REGION Network 6: Set SafetyGate Lock
   // 安全门锁定
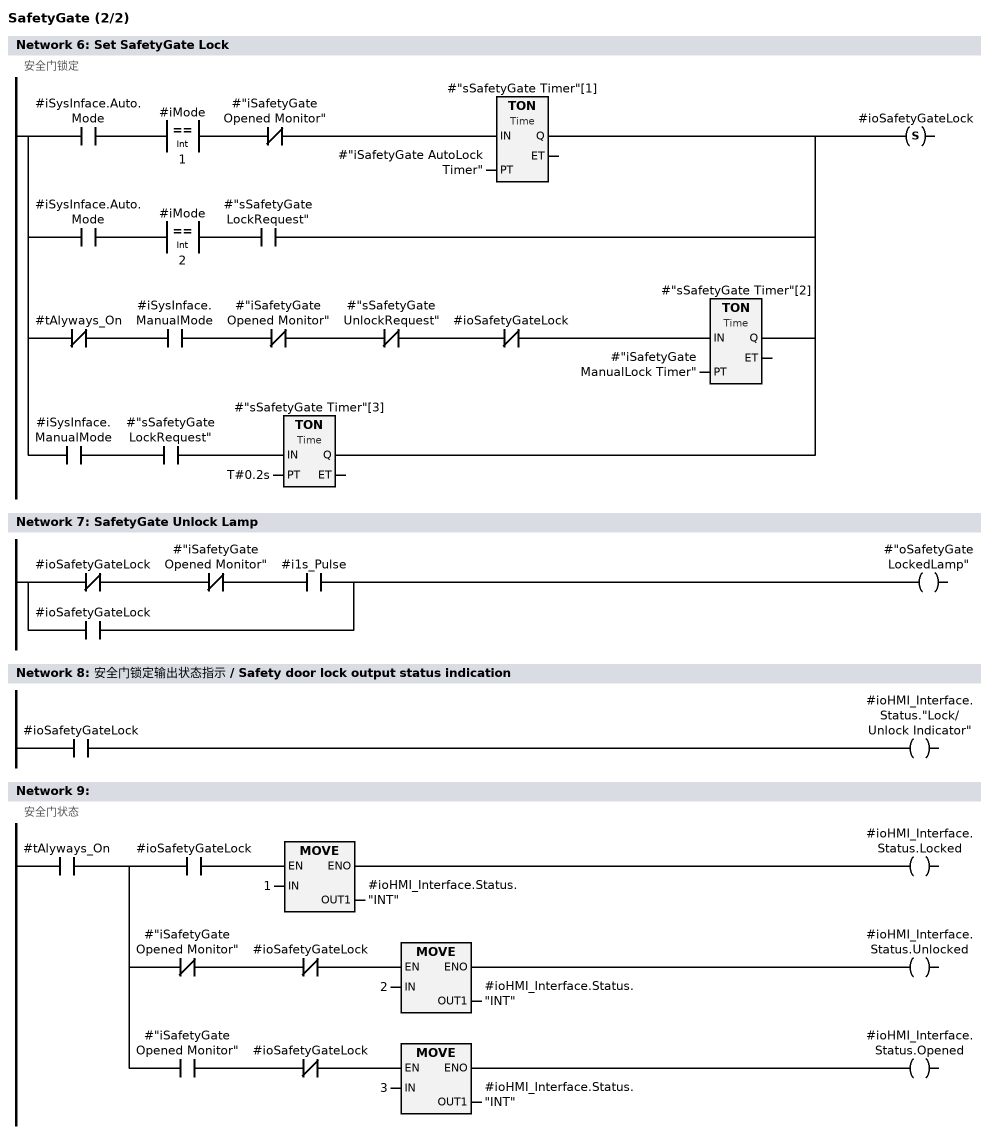
   RUNG wire#powerrail
      Contact( #iSysInface.Auto.Mode )
      { S7_Templates := "SrcType := Int" } EQ_Contact(in1 := #iMode, in2 := 1)
      I_Contact( #"iSafetyGate Opened Monitor" )
      { S7_Templates := "time_type := Time" } #"sSafetyGate Timer"[1].TON(pt := #"iSafetyGate AutoLock Timer", et =>)
      wire#w1
      S_Coil( #ioSafetyGateLock )
   END_RUNG
   RUNG wire#powerrail
      Contact( #iSysInface.Auto.Mode )
      { S7_Templates := "SrcType := Int" } EQ_Contact(in1 := #iMode, in2 := 2)
      Contact( #"sSafetyGate LockRequest" )
   END_RUNG wire#w1
   RUNG wire#powerrail
      I_Contact( #tAlyways_On )
      Contact( #iSysInface.ManualMode )
      I_Contact( #"iSafetyGate Opened Monitor" )
      I_Contact( #"sSafetyGate UnlockRequest" )
      I_Contact( #ioSafetyGateLock )
      { S7_Templates := "time_type := Time" } #"sSafetyGate Timer"[2].TON(pt := #"iSafetyGate ManualLock Timer", et =>)
   END_RUNG wire#w1
   RUNG wire#powerrail
      Contact( #iSysInface.ManualMode )
      Contact( #"sSafetyGate LockRequest" )
      { S7_Templates := "time_type := Time" } #"sSafetyGate Timer"[3].TON(pt := T#0.2s, et =>)
   END_RUNG wire#w1
   // the same network as SCL:
   #"sSafetyGate Timer"[1].TON(IN := #iSysInface.Auto.Mode AND (#iMode = 1) AND NOT #"iSafetyGate Opened Monitor",
                           PT := #"iSafetyGate AutoLock Timer");
   #_w1 := #"sSafetyGate Timer"[1].Q;
   #"sSafetyGate Timer"[2].TON(IN := NOT #tAlyways_On AND #iSysInface.ManualMode AND NOT #"iSafetyGate Opened Monitor" AND NOT #"sSafetyGate UnlockRequest" AND NOT #ioSafetyGateLock,
                           PT := #"iSafetyGate ManualLock Timer");
   #_w2 := #"sSafetyGate Timer"[2].Q;
   #"sSafetyGate Timer"[3].TON(IN := #iSysInface.ManualMode AND #"sSafetyGate LockRequest", PT := T#0.2s);
   IF #_w1 OR (#iSysInface.Auto.Mode AND (#iMode = 2) AND #"sSafetyGate LockRequest") OR #_w2 OR #"sSafetyGate Timer"[3].Q THEN
       #ioSafetyGateLock := TRUE;
   END_IF;
END_REGION

REGION Network 7: SafetyGate Unlock Lamp
   RUNG wire#powerrail
      I_Contact( #ioSafetyGateLock )
      I_Contact( #"iSafetyGate Opened Monitor" )
      Contact( #i1s_Pulse )
      wire#w1
      Coil( #"oSafetyGate LockedLamp" )
   END_RUNG
   RUNG wire#powerrail
      Contact( #ioSafetyGateLock )
   END_RUNG wire#w1
   // the same network as SCL:
   #"oSafetyGate LockedLamp" := (NOT #ioSafetyGateLock AND NOT #"iSafetyGate Opened Monitor" AND #i1s_Pulse) OR #ioSafetyGateLock;
END_REGION

REGION Network 8: 安全门锁定输出状态指示 / Safety door lock output status indication
   RUNG wire#powerrail
      Contact( #ioSafetyGateLock )
      Coil( #ioHMI_Interface.Status."Lock/Unlock Indicator" )
   END_RUNG
   // the same network as SCL:
   #ioHMI_Interface.Status."Lock/Unlock Indicator" := #ioSafetyGateLock;
END_REGION

REGION Network 9
   // 安全门状态
   RUNG wire#powerrail
      Contact( #tAlyways_On )
      wire#w1
      Contact( #ioSafetyGateLock )
      Move(in := 1, out1 => #ioHMI_Interface.Status."INT")
      Coil( #ioHMI_Interface.Status.Locked )
   END_RUNG
   RUNG wire#w1
      I_Contact( #"iSafetyGate Opened Monitor" )
      I_Contact( #ioSafetyGateLock )
      Move(in := 2, out1 => #ioHMI_Interface.Status."INT")
      Coil( #ioHMI_Interface.Status.Unlocked )
   END_RUNG
   RUNG wire#w1
      Contact( #"iSafetyGate Opened Monitor" )
      I_Contact( #ioSafetyGateLock )
      Move(in := 3, out1 => #ioHMI_Interface.Status."INT")
      Coil( #ioHMI_Interface.Status.Opened )
   END_RUNG
   // the same network as SCL:
   #_w1 := #tAlyways_On AND #ioSafetyGateLock;
   IF #_w1 THEN #ioHMI_Interface.Status."INT" := 1; END_IF;
   #ioHMI_Interface.Status.Locked := #_w1;
   #_w2 := #tAlyways_On AND NOT #"iSafetyGate Opened Monitor" AND NOT #ioSafetyGateLock;
   IF #_w2 THEN #ioHMI_Interface.Status."INT" := 2; END_IF;
   #ioHMI_Interface.Status.Unlocked := #_w2;
   #_w3 := #tAlyways_On AND #"iSafetyGate Opened Monitor" AND NOT #ioSafetyGateLock;
   IF #_w3 THEN #ioHMI_Interface.Status."INT" := 3; END_IF;
   #ioHMI_Interface.Status.Opened := #_w3;
END_REGION
END_FUNCTION_BLOCK

FUNCTION "ST10_PartData" : Void   // FC1500, SCL
{ S7_Optimized_Access := 'TRUE' }
// stored: SetENOAutomatically false
   VAR_INPUT
      iSysMode : "RCS_SysComInterface_V1";
   END_VAR
   VAR_TEMP
      idex : Int;
   END_VAR
BEGIN
END_FUNCTION

FUNCTION "ST10_Analog" : Void   // FC1080, SCL
{ S7_Optimized_Access := 'TRUE' }
// stored: AutoNumber false, SetENOAutomatically false
   VAR_INPUT
      iSysMode : "RCS_SysComInterface_V1";
   END_VAR
   VAR_TEMP
      idex : Int;
   END_VAR
BEGIN


   REGION 氮气压模拟量
       //定义编号
       #idex := 1;
       //功能块调用

    END_REGION
END_FUNCTION

FUNCTION "CuringOven" : Void   // FC900, LAD
{ S7_Optimized_Access := 'TRUE' }
// stored: AutoNumber false, SetENOAutomatically false
BEGIN

REGION Network 1
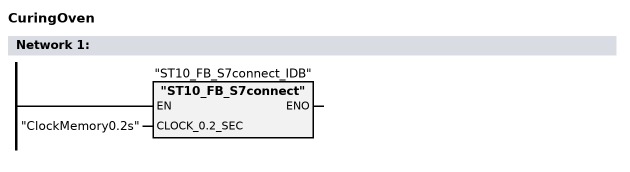
   RUNG wire#powerrail
      "ST10_FB_S7connect_IDB"("CLOCK_0.2_SEC" := "ClockMemory0.2s")
   END_RUNG
   // the same network as SCL:
   "ST10_FB_S7connect_IDB"("CLOCK_0.2_SEC" := "ClockMemory0.2s");   // "ST10_FB_S7connect"
END_REGION
END_FUNCTION

FUNCTION_BLOCK "ST10_FB_S7connect"   // FB900, LAD
{ S7_Optimized_Access := 'TRUE' }
VERSION : 0.1
// stored: AutoNumber false, IsIECCheckEnabled false, IsRetainMemResEnabled false, MemoryReserve 100, SetENOAutomatically false, UDAEnableTagReadback false
   VAR_INPUT
      "CLOCK_0.2_SEC" : Bool;
   END_VAR
   VAR
      Always_On : Bool;
      Status_Get : Array[1..6] of Struct
         NDR : Bool;
         Error : Bool;
         Status : Int;
      END_STRUCT;
      Status_Put : Array[1..6] of Struct
         Done : Bool;
         Error : Bool;
         Status : Int;
      END_STRUCT;
      GET_Instance1 { S7_SetPoint := 'True'} : GET;
      GET_Instance2 { S7_SetPoint := 'True'} : GET;
      PUT_Instance1 { S7_SetPoint := 'True'} : PUT;
      PUT_Instance2 { S7_SetPoint := 'True'} : PUT;
      PLs { S7_SetPoint := 'True'} : Array[1..6] of Bool;
   END_VAR
   VAR DB_SPECIFIC
      TON : Array[1..5] of TON_TIME;
   END_VAR
   VAR
      NextStation_OffLine : Bool;   // S7心跳超时
   END_VAR
BEGIN

REGION Network 1: **************** 和40交互 **************** / **************** ****************
END_REGION

REGION Network 2: PUT
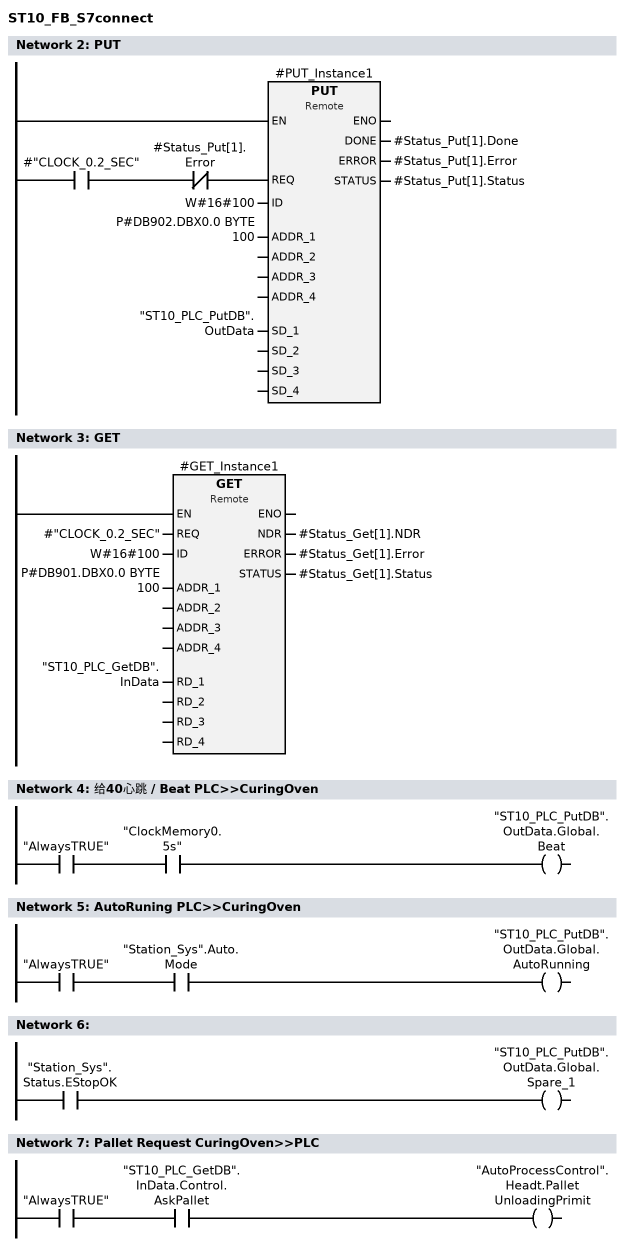
   RUNG wire#powerrail
      { S7_Templates := "[remote_type := Remote, local_type := Variant]" } #PUT_Instance1.PUT(REQ := wire#w1, ID := W#16#100, ADDR_1 := P#DB902.DBX0.0 BYTE 100, ADDR_2 :=, ADDR_3 :=, ADDR_4 :=, SD_1 := "ST10_PLC_PutDB".OutData, SD_2 :=, SD_3 :=, SD_4 :=, DONE => #Status_Put[1].Done, ERROR => #Status_Put[1].Error, STATUS => #Status_Put[1].Status)
   END_RUNG
   RUNG wire#powerrail
      Contact( #"CLOCK_0.2_SEC" )
      I_Contact( #Status_Put[1].Error )
   END_RUNG wire#w1
   // the same network as SCL:
   #PUT_Instance1(REQ := #"CLOCK_0.2_SEC" AND NOT #Status_Put[1].Error,   // PUT
                  ID := W#16#100,
                  ADDR_1 := P#DB902.DBX0.0 BYTE 100,
                  SD_1 := "ST10_PLC_PutDB".OutData,
                  DONE => #Status_Put[1].Done,
                  ERROR => #Status_Put[1].Error,
                  STATUS => #Status_Put[1].Status);
END_REGION

REGION Network 3: GET
   RUNG wire#powerrail
      { S7_Templates := "[remote_type := Remote, local_type := Variant]" } #GET_Instance1.GET(REQ := #"CLOCK_0.2_SEC", ID := W#16#100, ADDR_1 := P#DB901.DBX0.0 BYTE 100, ADDR_2 :=, ADDR_3 :=, ADDR_4 :=, RD_1 := "ST10_PLC_GetDB".InData, RD_2 :=, RD_3 :=, RD_4 :=, NDR => #Status_Get[1].NDR, ERROR => #Status_Get[1].Error, STATUS => #Status_Get[1].Status)
   END_RUNG
   // the same network as SCL:
   #GET_Instance1(REQ := #"CLOCK_0.2_SEC",   // GET
                  ID := W#16#100,
                  ADDR_1 := P#DB901.DBX0.0 BYTE 100,
                  RD_1 := "ST10_PLC_GetDB".InData,
                  NDR => #Status_Get[1].NDR,
                  ERROR => #Status_Get[1].Error,
                  STATUS => #Status_Get[1].Status);
END_REGION

REGION Network 4: 给40心跳 / Beat PLC>>CuringOven
   RUNG wire#powerrail
      Contact( "AlwaysTRUE" )
      Contact( "ClockMemory0.5s" )
      Coil( "ST10_PLC_PutDB".OutData.Global.Beat )
   END_RUNG
   // the same network as SCL:
   "ST10_PLC_PutDB".OutData.Global.Beat := "AlwaysTRUE" AND "ClockMemory0.5s";
END_REGION

REGION Network 5: AutoRuning PLC>>CuringOven
   RUNG wire#powerrail
      Contact( "AlwaysTRUE" )
      Contact( "Station_Sys".Auto.Mode )
      Coil( "ST10_PLC_PutDB".OutData.Global.AutoRunning )
   END_RUNG
   // the same network as SCL:
   "ST10_PLC_PutDB".OutData.Global.AutoRunning := "AlwaysTRUE" AND "Station_Sys".Auto.Mode;
END_REGION

REGION Network 6
   RUNG wire#powerrail
      Contact( "Station_Sys".Status.EStopOK )
      Coil( "ST10_PLC_PutDB".OutData.Global.Spare_1 )
   END_RUNG
   // the same network as SCL:
   "ST10_PLC_PutDB".OutData.Global.Spare_1 := "Station_Sys".Status.EStopOK;
END_REGION

REGION Network 7: Pallet Request CuringOven>>PLC
   RUNG wire#powerrail
      Contact( "AlwaysTRUE" )
      Contact( "ST10_PLC_GetDB".InData.Control.AskPallet )
      Coil( "AutoProcessControl".Headt.PalletUnloadingPrimit )
   END_RUNG
   // the same network as SCL:
   "AutoProcessControl".Headt.PalletUnloadingPrimit := "AlwaysTRUE" AND "ST10_PLC_GetDB".InData.Control.AskPallet;
END_REGION
END_FUNCTION_BLOCK

FUNCTION "IV3" : Void   // FC2100, LAD
{ S7_Optimized_Access := 'TRUE' }
VERSION : 0.1
// stored: AutoNumber false, IsIECCheckEnabled false, SetENOAutomatically false, UDAEnableTagReadback false
BEGIN

REGION Network 1: IV3
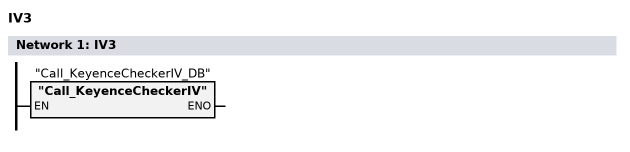
   RUNG wire#powerrail
      "Call_KeyenceCheckerIV_DB"()
   END_RUNG
   // the same network as SCL:
   "Call_KeyenceCheckerIV_DB"();   // "Call_KeyenceCheckerIV"
END_REGION
END_FUNCTION

FUNCTION_BLOCK "Call_KeyenceCheckerIV"   // FB2100, SCL
{ S7_Optimized_Access := 'TRUE' }
// stored: AutoNumber false, MemoryReserve 100, SetENOAutomatically false
   VAR
      InsKeyenceCheckerIV3810A1 : "FB_KeyenceCheckerIV3";   // 声明相机功能块的实例
      InsKeyenceCheckerIV3811A1 : "FB_KeyenceCheckerIV3";   // 声明相机功能块的实例
      nIndex { S7_SetPoint := 'True'} : Int;
   END_VAR
BEGIN

   //810A1
   REGION KeyenceCheckerIV3() 

       REGION HardwareConfigGuidance()
           // 组态说明/Hardware config Guidance
           // 输入/Input
           // Command Status Bits_1
           // Device Result Bits_1
           // Device Status Words_1
           // Device Statistics_1
           // Position Adjust Result_1
           // Tool Result_1
           // Tool Result_2
           // 输出/Output
           // Command Control_1
       END_REGION

       REGION DeviceControl()
           //************************************************************************************************ 
           //设备控制/Device control 
           //************************************************************************************************ 
           //Set device number
           #nIndex := 1;//(For example Constant:ST01_CHECKER_FUNCTION)

           REGION WorkflowControl()
               //************************************************************************************************ 
               //流程控制/Workflow control
               //************************************************************************************************ 
               //---set program number
               //   "DB_KeyenceCheckerIV2".aDev[#nIndex].Out.CommandControl.nProgramNo
               //---set command mode and wait for mode to "MODE_CHECKER_IDLE"
               //   "DB_KeyenceCheckerIV2".aDev[#nIndex].Common.nMode
           END_REGION

           REGION GeneralControl()
               //************************************************************************************************ 
               //常规控制/General control 
               //************************************************************************************************ 
               //Set common parameter
               "DB_KeyenceCheckerIV3".aDev[#nIndex].Common.bScreenActive := "Station_Sys".Manual.Mode;
               "DB_KeyenceCheckerIV3".aDev[#nIndex].Common.bReset := "Station_Sys".Cmd.Reset;
               "DB_KeyenceCheckerIV3".aDev[#nIndex].Common.tMaxProcessTime := t#30s;
           END_REGION

           REGION ParameterConfig()
               //************************************************************************************************ 
               //参数配置/Parameter config 
               //************************************************************************************************ 
           END_REGION

           REGION ModeControl()
               //************************************************************************************************ 
               //设备启动停止/Device mode control
               //************************************************************************************************ 
               // IF NOT "Station_Sys".Status.Run THEN
               //     "DB_KeyenceCheckerIV3".aDev[#nIndex].Common.nMode := 0;
               // END_IF;

               IF "Station_Sys".Manual.Mode THEN
                   "DB_KeyenceCheckerIV3".aDev[#nIndex].Common.nModeSwitch := "MS_MANUAL";
               ELSIF "Station_Sys".Auto.Mode THEN
                   "DB_KeyenceCheckerIV3".aDev[#nIndex].Common.nModeSwitch:=  "MS_Auto";
               ELSE
                   "DB_KeyenceCheckerIV3".aDev[#nIndex].Common.nModeSwitch := "MS_EMPTY";
               END_IF;
               END_REGION

           REGION ConditionControl()
               //************************************************************************************************ 
               //使能控制/Condition control
               //************************************************************************************************ 
               //according to detail information in different use to fill in start condition
               "DB_KeyenceCheckerIV3".aDev[#nIndex].Common.bEnable := "Station_Sys".Status.Run;
           END_REGION

       END_REGION

       REGION HardwareInput()
           //************************************************************************************************ 
           //硬件输入/Hardware input 
           //************************************************************************************************ 
       END_REGION

       REGION CallFunctionBlock()
           //************************************************************************************************
           //功能块调用/Call function block
           //************************************************************************************************
           //according to hardware configuration to type in hardware address

           #InsKeyenceCheckerIV3810A1(#nIndex);


       END_REGION

       REGION HardwareOutput()
           //************************************************************************************************ 
           //硬件输出/Hardware output 
           //************************************************************************************************ 
       END_REGION

   END_REGION


   //811A1
   REGION KeyenceCheckerIV3() 

       REGION HardwareConfigGuidance()
           // 组态说明/Hardware config Guidance
           // 输入/Input
           // Command Status Bits_1
           // Device Result Bits_1
           // Device Status Words_1
           // Device Statistics_1
           // Position Adjust Result_1
           // Tool Result_1
           // Tool Result_2
           // 输出/Output
           // Command Control_1
       END_REGION

       REGION DeviceControl()
           //************************************************************************************************ 
           //设备控制/Device control 
           //************************************************************************************************ 
           //Set device number
           #nIndex := 2;//(For example Constant:ST01_CHECKER_FUNCTION)

           REGION WorkflowControl()
               //************************************************************************************************ 
               //流程控制/Workflow control
               //************************************************************************************************ 
               //---set program number
               //   "DB_KeyenceCheckerIV2".aDev[#nIndex].Out.CommandControl.nProgramNo
               //---set command mode and wait for mode to "MODE_CHECKER_IDLE"
               //   "DB_KeyenceCheckerIV2".aDev[#nIndex].Common.nMode
           END_REGION

           REGION GeneralControl()
               //************************************************************************************************ 
               //常规控制/General control 
               //************************************************************************************************ 
               //Set common parameter
               "DB_KeyenceCheckerIV3".aDev[#nIndex].Common.bScreenActive := "Station_Sys".Manual.Mode;
               "DB_KeyenceCheckerIV3".aDev[#nIndex].Common.bReset := "Station_Sys".Cmd.Reset;
               "DB_KeyenceCheckerIV3".aDev[#nIndex].Common.tMaxProcessTime := t#30s;
           END_REGION

           REGION ParameterConfig()
               //************************************************************************************************ 
               //参数配置/Parameter config 
               //************************************************************************************************ 
           END_REGION

           REGION ModeControl()
               //************************************************************************************************ 
               //设备启动停止/Device mode control
               //************************************************************************************************ 
               // IF NOT "Station_Sys".Status.Run THEN
               //     "DB_KeyenceCheckerIV3".aDev[#nIndex].Common.nMode := 0;
               // END_IF;

               IF "Station_Sys".Manual.Mode THEN
                   "DB_KeyenceCheckerIV3".aDev[#nIndex].Common.nModeSwitch := "MS_MANUAL";
               ELSIF "Station_Sys".Auto.Mode THEN
                   "DB_KeyenceCheckerIV3".aDev[#nIndex].Common.nModeSwitch := "MS_Auto";
               ELSE
                   "DB_KeyenceCheckerIV3".aDev[#nIndex].Common.nModeSwitch := "MS_EMPTY";
               END_IF;
           END_REGION

           REGION ConditionControl()
               //************************************************************************************************ 
               //使能控制/Condition control
               //************************************************************************************************ 
               //according to detail information in different use to fill in start condition
               "DB_KeyenceCheckerIV3".aDev[#nIndex].Common.bEnable := "Station_Sys".Status.Run;
           END_REGION

       END_REGION

       REGION HardwareInput()
           //************************************************************************************************ 
           //硬件输入/Hardware input 
           //************************************************************************************************ 
       END_REGION

       REGION CallFunctionBlock()
           //************************************************************************************************
           //功能块调用/Call function block
           //************************************************************************************************
           //according to hardware configuration to type in hardware address

           #InsKeyenceCheckerIV3811A1(#nIndex);


       END_REGION

       REGION HardwareOutput()
           //************************************************************************************************ 
           //硬件输出/Hardware output 
           //************************************************************************************************ 
       END_REGION

   END_REGION
END_FUNCTION_BLOCK

FUNCTION "IAI" : Void   // FC2200, LAD
{ S7_Optimized_Access := 'TRUE' }
// stored: AutoNumber false, SetENOAutomatically false
BEGIN

REGION Network 1 (SCL): 模式 / Mode
   "ModeDB".Gen.Out.Estop := "Station_Sys".Status.EStopOK;
   "ModeDB".Gen.Out.Reset := "Station_Sys".Cmd.Reset;
   "ModeDB".Gen.Out.Manual := "Station_Sys".Manual.Mode;
   "ModeDB".Gen.Out.Auto := "Station_Sys".Auto.Mode;
   "ModeDB".Gen.Out.Home := "Station_Sys".Initial.Running;
   "ModeDB".Gen.Out.Running := "Station_Sys".Auto.Mode;//"Station_Sys".Auto.Running OR "ST10_PM".Num[7].InitialRun;
   //"ModeDB".Gen.Out.Change:=
END_REGION

REGION Network 2
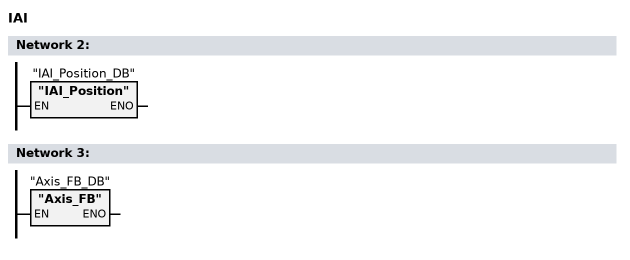
   RUNG wire#powerrail
      "IAI_Position_DB"()
   END_RUNG
   // the same network as SCL:
   "IAI_Position_DB"();   // "IAI_Position"
END_REGION

REGION Network 3
   RUNG wire#powerrail
      "Axis_FB_DB"()
   END_RUNG
   // the same network as SCL:
   "Axis_FB_DB"();   // "Axis_FB"
END_REGION
END_FUNCTION

FUNCTION_BLOCK "IAI_Position"   // FB2210, LAD
{ S7_Optimized_Access := 'TRUE' }
// stored: AutoNumber false, MemoryReserve 100, SetENOAutomatically false
   VAR
      Servo5 { S7_SetPoint := 'True'} : "SevroStart&PosCheck_IAI";
      Servo6 { S7_SetPoint := 'True'} : "SevroStart&PosCheck_IAI";
      Servo7 { S7_SetPoint := 'True'} : "SevroStart&PosCheck_IAI";
   END_VAR
   VAR_TEMP
      Sevro5ActPos : Real;
      Sevro5StartList : Bool;
      Sevro6ActPos : Real;
      Sevro6StartList : Bool;
      Sevro7ActPos : Real;
      Sevro7StartList : Bool;
   END_VAR
BEGIN

REGION Network 2 (SCL)
   REGION Servo position judgment
       FOR "IAI_DeviceCtl".IAIServo[1].i := 1 TO 12 BY 1 DO
           "IAI_DeviceCtl".IAIServo[1].Pos.List["IAI_DeviceCtl".IAIServo[1].i].Pos := "IAI_A1".Auto.Pos["IAI_DeviceCtl".IAIServo[1].i].Pos;
           "IAI_DeviceCtl".IAIServo[1].Pos.List["IAI_DeviceCtl".IAIServo[1].i].Vel := "IAI_A1".Auto.Pos["IAI_DeviceCtl".IAIServo[1].i].Vel;

           "IAI_DeviceCtl".IAIServo[2].Pos.List["IAI_DeviceCtl".IAIServo[1].i].Pos := "IAI_A2".Auto.Pos["IAI_DeviceCtl".IAIServo[1].i].Pos;
           "IAI_DeviceCtl".IAIServo[2].Pos.List["IAI_DeviceCtl".IAIServo[1].i].Vel := "IAI_A2".Auto.Pos["IAI_DeviceCtl".IAIServo[1].i].Vel;

           "IAI_DeviceCtl".IAIServo[3].Pos.List["IAI_DeviceCtl".IAIServo[1].i].Pos := "IAI_A3".Auto.Pos["IAI_DeviceCtl".IAIServo[1].i].Pos;
           "IAI_DeviceCtl".IAIServo[3].Pos.List["IAI_DeviceCtl".IAIServo[1].i].Vel := "IAI_A3".Auto.Pos["IAI_DeviceCtl".IAIServo[1].i].Vel;


       END_FOR;

       (******************************************************* SV1 Z轴 ********************************************************************)
       //伺服位置判断
       #"Servo5"(iRef_Homed := 1,
                 iStandstill := FALSE,
                 iReset := "Station_Sys".Cmd.Reset,
                 interlcok := 1,
                 "iActual Posi" := "Axis_FB_DB".IAI_Axis[1].CurrentPosition,
                 "iTol+" := 0.5,
                 "iTol-" := 0.5,
                 iStartTon := T#100mS,
                 ioPoint := "IAI_DeviceCtl".IAIServo[1].Point,
                 oStartPos => #Sevro5StartList,
                 ioList := "IAI_DeviceCtl".IAIServo[1].Pos,
                 ioPosNumberSelect := "IAI_DeviceCtl".IAIServo[1].nPositionListNo);

       IF "IAI_DeviceCtl".IAIServo[1].nPositionListNo = 0 THEN
           "IAI_DeviceCtl".IAIServo[1].nPositionListNo := 1;
       END_IF;

       "Axis_FB_DB".IAI_Axis[1].Par.PosCode:="IAI_A1".Auto.Index := "IAI_DeviceCtl".IAIServo[1].nPositionListNo;

       //伺服启动
       "IAI_A1".In.iAutoStart := #Sevro5StartList AND "Station_Sys".Auto.Mode;

       (******************************************************* SV2 X轴********************************************************************)
       //伺服位置判断
       #"Servo6"(iRef_Homed := 1,
                 iStandstill := FALSE,
                 iReset := "Station_Sys".Cmd.Reset,
                 interlcok := 1,
                 "iActual Posi" := "Axis_FB_DB".IAI_Axis[2].CurrentPosition,
                 "iTol+" := 0.5,
                 "iTol-" := 0.5,
                 iStartTon := T#100mS,
                 ioPoint := "IAI_DeviceCtl".IAIServo[2].Point,
                 oStartPos => #Sevro6StartList,
                 ioList := "IAI_DeviceCtl".IAIServo[2].Pos,
                 ioPosNumberSelect := "IAI_DeviceCtl".IAIServo[2].nPositionListNo);

       IF "IAI_DeviceCtl".IAIServo[2].nPositionListNo = 0 THEN
           "IAI_DeviceCtl".IAIServo[2].nPositionListNo := 1;
       END_IF;

       "Axis_FB_DB".IAI_Axis[2].Par.PosCode:="IAI_A2".Auto.Index := "IAI_DeviceCtl".IAIServo[2].nPositionListNo;

       //伺服启动
       "IAI_A2".In.iAutoStart := #Sevro6StartList AND "Station_Sys".Auto.Mode;

       (******************************************************* SV3 Y轴********************************************************************)
       //伺服位置判断
       #"Servo7"(iRef_Homed := 1,
                 iStandstill := FALSE,
                 iReset := "Station_Sys".Cmd.Reset,
                 interlcok := 1,
                 "iActual Posi" := "Axis_FB_DB".IAI_Axis[3].CurrentPosition,
                 "iTol+" := 0.5,
                 "iTol-" := 0.5,
                 iStartTon := T#100mS,
                 ioPoint := "IAI_DeviceCtl".IAIServo[3].Point,
                 oStartPos => #Sevro7StartList,
                 ioList := "IAI_DeviceCtl".IAIServo[3].Pos,
                 ioPosNumberSelect := "IAI_DeviceCtl".IAIServo[3].nPositionListNo);

       IF "IAI_DeviceCtl".IAIServo[3].nPositionListNo = 0 THEN
           "IAI_DeviceCtl".IAIServo[3].nPositionListNo := 1;
       END_IF;

       "Axis_FB_DB".IAI_Axis[3].Par.PosCode:="IAI_A3".Auto.Index := "IAI_DeviceCtl".IAIServo[3].nPositionListNo;

       //伺服启动
       "IAI_A3".In.iAutoStart := #Sevro7StartList AND "Station_Sys".Auto.Mode;
   END_REGION
END_REGION
END_FUNCTION_BLOCK

FUNCTION_BLOCK "SevroStart&PosCheck_IAI"   // FB2209, LAD
{ S7_Optimized_Access := 'TRUE' }
// stored: AutoNumber false, MemoryReserve 100, SetENOAutomatically false
   VAR_INPUT
      iRef_Homed { ExternalAccessible := 'False'; ExternalVisible := 'False'; ExternalWritable := 'False'} : Bool;
      iStandstill { ExternalAccessible := 'False'; ExternalVisible := 'False'; ExternalWritable := 'False'} : Bool;
      iReset : Bool;
      interlcok : Bool;   // 启动互锁
      "iActual Posi" { ExternalAccessible := 'False'; ExternalVisible := 'False'; ExternalWritable := 'False'} : Real;
      "iTol+" { ExternalAccessible := 'False'; ExternalVisible := 'False'; ExternalWritable := 'False'} : Real;
      "iTol-" { ExternalAccessible := 'False'; ExternalVisible := 'False'; ExternalWritable := 'False'} : Real;
      iStartTon : Time := T#200ms;   // 启动延迟
   END_VAR
   VAR_OUTPUT
      oStartPos : Bool;   // 启动
      DoublePosError : Bool;   // 多位置触发
   END_VAR
   VAR_IN_OUT
      ioPoint : Array[0..39] of Struct
         Start : Bool;
         Achieve : Bool;
      END_STRUCT;
      ioList : "PosList_IAI";
      ioPosNumberSelect : Int;   // 位置启动
   END_VAR
   VAR
      TON : Array[0..1] of TON_TIME;
      StartCount { S7_SetPoint := 'True'} : Int;   // 启动计数
   END_VAR
   VAR_TEMP
      "Actual Posi+Tol" : Real;
      "Actual Posi-Tol" : Real;
      Index : Array[0..7] of Int;   // 位置启动
      PosStart : Bool;
   END_VAR
   VAR_TEMP   // added for the SCL form of the ladder/FBD networks
      _w1 : Bool;
   END_VAR
BEGIN

REGION Network 1 (SCL): 检查当前启动位置号
   #Index[1] := 0;
   #PosStart := false;
   FOR #Index[1] := 0 TO 39 DO
       IF #ioPoint[#Index[1]].Start THEN

           #ioPosNumberSelect := #Index[1];//当前启动位置号
           #PosStart := TRUE;
           EXIT;
       END_IF;
   END_FOR;
   #Index[2] := 0;
   #StartCount := 0;
   FOR #Index[2] := 0 TO 39 DO
       IF #ioPoint[#Index[2]].Start THEN

           #StartCount := #StartCount+1;//当前启动位置号


       END_IF;
       IF #Index[2] = 39 THEN

           EXIT;
       END_IF;

   END_FOR;
END_REGION

REGION Network 2: 位置给定
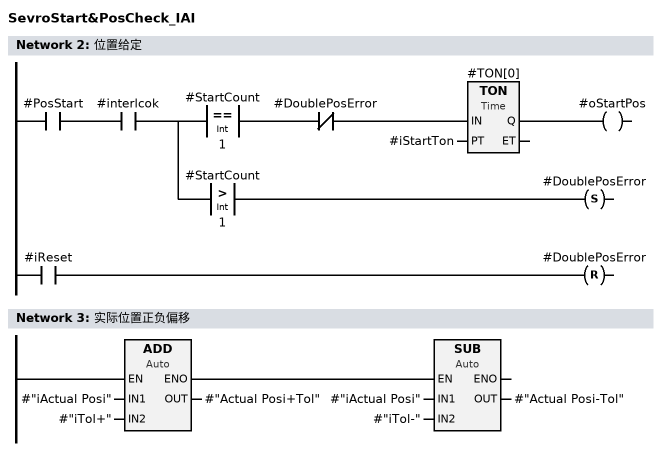
   RUNG wire#powerrail
      Contact( #PosStart )
      Contact( #interlcok )
      wire#w1
      { S7_Templates := "SrcType := Int" } EQ_Contact(in1 := #StartCount, in2 := 1)
      I_Contact( #DoublePosError )
      { S7_Templates := "time_type := Time" } #TON[0].TON(pt := #iStartTon, et =>)
      Coil( #oStartPos )
   END_RUNG
   RUNG wire#w1
      { S7_Templates := "SrcType := Int" } GT_Contact(in1 := #StartCount, in2 := 1)
      S_Coil( #DoublePosError )
   END_RUNG
   RUNG wire#powerrail
      Contact( #iReset )
      R_Coil( #DoublePosError )
   END_RUNG
   // the same network as SCL:
   #_w1 := #PosStart AND #interlcok;
   #TON[0].TON(IN := #_w1 AND (#StartCount = 1) AND NOT #DoublePosError, PT := #iStartTon);
   #oStartPos := #TON[0].Q;
   IF #_w1 AND (#StartCount > 1) THEN #DoublePosError := TRUE; END_IF;
   IF #iReset THEN #DoublePosError := FALSE; END_IF;
END_REGION

REGION Network 3: 实际位置正负偏移
   RUNG wire#powerrail
      Add(in1 := #"iActual Posi", in2 := #"iTol+", out => #"Actual Posi+Tol")
      Sub(in1 := #"iActual Posi", in2 := #"iTol-", out => #"Actual Posi-Tol")
   END_RUNG
   // the same network as SCL:
   #"Actual Posi+Tol" := #"iActual Posi" + #"iTol+";
   #"Actual Posi-Tol" := #"iActual Posi" - #"iTol-";
END_REGION

REGION Network 4 (SCL): 位置检查


   #Index[3] := 0;
   FOR #Index[3] := 0 TO 39 DO
       IF #ioList.List[ #Index[3]].Pos>= #"Actual Posi-Tol"
           AND #ioList.List[ #Index[3]].Pos<= #"Actual Posi+Tol"
       THEN
         #ioPoint[#Index[3]].Achieve := TRUE;
       ELSE
           #ioPoint[#Index[3]].Achieve := FALSE;
       END_IF;
   END_FOR;
END_REGION
END_FUNCTION_BLOCK

FUNCTION_BLOCK "Axis_FB"   // FB2200, SCL
{ S7_Optimized_Access := 'FALSE' }
// stored: AutoNumber false, SetENOAutomatically false
   VAR
      IAI_Axis { S7_SetPoint := 'True'} : Array[1..3] of "IAI_BASE_FB";
   END_VAR
   VAR CONSTANT
      Z_Axis : Int := 1;
      Y_axis : Int := 3;
      X_Axis : Int := 2;
   END_VAR
BEGIN
   ///Z轴

   #IAI_Axis[X_Axis].Enable := #IAI_Axis[Y_axis].Enable := #IAI_Axis[Z_Axis].Enable := "ST10_SystemModeFB_iDB".iEstopAllOK AND "ST10_SystemModeFB_iDB".iSafetyDoor;

   #IAI_Axis[Z_Axis]();

   #IAI_Axis[Z_Axis].Axis_ID := 1;
   #IAI_Axis[Z_Axis]."Input 4 word_Man1" := "OP10_384A1~Input_4_word_7";
   #IAI_Axis[Z_Axis]."Input 4 word_Man2" := "OP10_384A1~Input_4_word_8";
   #IAI_Axis[Z_Axis]."Input 4 word_1" := "OP10_384A1~Input_4_word_3";
   #IAI_Axis[Z_Axis]."Input 4 word_2" := "OP10_384A1~Input_4_word_4";
   #IAI_Axis[Z_Axis]."Output 4 word_Man1" := "OP10_384A1~Output_4_word_1";
   #IAI_Axis[Z_Axis]."Output 4 word_Man2" := "OP10_384A1~Output_4_word_2";
   #IAI_Axis[Z_Axis]."Output 4 word_1" := "OP10_384A1~Output_4_word_5";
   #IAI_Axis[Z_Axis]."Output 4 word_2" := "OP10_384A1~Output_4_word_6";

   #IAI_Axis[Z_Axis].Mode:= "ModeDB".Gen;
   #IAI_Axis[Z_Axis].Par.PositionWidth := 0.05;
   #IAI_Axis[Z_Axis].Par.AccSpeed := 10;
   #IAI_Axis[Z_Axis].Par.DecSpeed := 10;
   #IAI_Axis[Z_Axis].Par."Limt+Pos" := 362000.0;
   #IAI_Axis[Z_Axis].Par."Limt-Pos" := -30000.0;
   #IAI_Axis[Z_Axis].Par.Speed:= 10;

   #IAI_Axis[Z_Axis].Interfere := TRUE;
   #IAI_Axis[Z_Axis].RunSetTime := T#20S;
   #IAI_Axis[Z_Axis].Par.GoPosInterfere[0] := TRUE;
   #IAI_Axis[Z_Axis].Par.GoPosInterfere[1] := TRUE;
   #IAI_Axis[Z_Axis].Par.GoPosInterfere[2] := TRUE;
   #IAI_Axis[Z_Axis].Par.GoPosInterfere[3] := TRUE;
   #IAI_Axis[Z_Axis].Par.GoPosInterfere[4] := TRUE;
   #IAI_Axis[Z_Axis].Par.GoPosInterfere[5] := TRUE;
   #IAI_Axis[Z_Axis].AutoPointStart := "IAI_A1".In.iAutoStart;

   "IAI_A1".Auto.Pos[1].Pos:=#IAI_Axis[Z_Axis].Par.TargetPosition[1] := "Parameter".AxisRun.Axis[5].Pos1.Position;
   "IAI_A1".Auto.Pos[1].Vel :=#IAI_Axis[Z_Axis].Par.TargetSpeed[1] := "Parameter".AxisRun.Axis[5].Pos1.Speed;

   "IAI_A1".Auto.Pos[2].Pos:=#IAI_Axis[Z_Axis].Par.TargetPosition[2] := "Parameter".AxisRun.Axis[5].Pos2.Position;
   "IAI_A1".Auto.Pos[2].Vel :=#IAI_Axis[Z_Axis].Par.TargetSpeed[2] := "Parameter".AxisRun.Axis[5].Pos2.Speed;

   "IAI_A1".Auto.Pos[3].Pos:=#IAI_Axis[Z_Axis].Par.TargetPosition[3] := "Parameter".AxisRun.Axis[5].Pos3.Position;
   "IAI_A1".Auto.Pos[3].Vel :=#IAI_Axis[Z_Axis].Par.TargetSpeed[3] := "Parameter".AxisRun.Axis[5].Pos3.Speed;

   "IAI_A1".Auto.Pos[4].Pos:=#IAI_Axis[Z_Axis].Par.TargetPosition[4] := "Parameter".AxisRun.Axis[5].Pos4.Position;
   "IAI_A1".Auto.Pos[4].Vel :=#IAI_Axis[Z_Axis].Par.TargetSpeed[4] := "Parameter".AxisRun.Axis[5].Pos4.Speed;

   "IAI_A1".Auto.Pos[5].Pos:=#IAI_Axis[Z_Axis].Par.TargetPosition[5] := "Parameter".AxisRun.Axis[5].Pos5.Position;
   "IAI_A1".Auto.Pos[5].Vel :=#IAI_Axis[Z_Axis].Par.TargetSpeed[5] := "Parameter".AxisRun.Axis[5].Pos5.Speed;

   "IAI_A1".Auto.Pos[6].Pos := #IAI_Axis[Z_Axis].Par.TargetPosition[6] := "Parameter".AxisRun.Axis[5].Pos6.Position;
   "IAI_A1".Auto.Pos[6].Vel := #IAI_Axis[Z_Axis].Par.TargetSpeed[6] := "Parameter".AxisRun.Axis[5].Pos6.Speed;

   "IAI_A1".Auto.Pos[7].Pos := #IAI_Axis[Z_Axis].Par.TargetPosition[7] := "Parameter".AxisRun.Axis[5].Pos7.Position;
   "IAI_A1".Auto.Pos[7].Vel := #IAI_Axis[Z_Axis].Par.TargetSpeed[7] := "Parameter".AxisRun.Axis[5].Pos7.Speed;

   "IAI_A1".Auto.Pos[8].Pos := #IAI_Axis[Z_Axis].Par.TargetPosition[8] := "Parameter".AxisRun.Axis[5].Pos8.Position;
   "IAI_A1".Auto.Pos[8].Vel := #IAI_Axis[Z_Axis].Par.TargetSpeed[8] := "Parameter".AxisRun.Axis[5].Pos8.Speed;

   "IAI_A1".Auto.Pos[9].Pos := #IAI_Axis[Z_Axis].Par.TargetPosition[9] := "Parameter".AxisRun.Axis[5].Pos6.Position-4.0;
   "IAI_A1".Auto.Pos[9].Vel := #IAI_Axis[Z_Axis].Par.TargetSpeed[9] := "Parameter".AxisRun.Axis[5].Pos6.Speed;

   "IAI_A1".Auto.Pos[10].Pos := #IAI_Axis[Z_Axis].Par.TargetPosition[10] := "Parameter".AxisRun.Axis[5].Pos10.Position;
   "IAI_A1".Auto.Pos[10].Vel := #IAI_Axis[Z_Axis].Par.TargetSpeed[10] := "Parameter".AxisRun.Axis[5].Pos10.Speed;

   //X轴
   #IAI_Axis[X_Axis]();

   #IAI_Axis[X_Axis].Axis_ID := 2;
   #IAI_Axis[X_Axis]."Input 4 word_Man1" := "OP10_384A1~Input_4_word_7";
   #IAI_Axis[X_Axis]."Input 4 word_Man2" := "OP10_384A1~Input_4_word_8";
   #IAI_Axis[X_Axis]."Input 4 word_1" := "OP10_384A1~Input_4_word_5";
   #IAI_Axis[X_Axis]."Input 4 word_2" := "OP10_384A1~Input_4_word_6";
   #IAI_Axis[X_Axis]."Output 4 word_Man1" := "OP10_384A1~Output_4_word_1";
   #IAI_Axis[X_Axis]."Output 4 word_Man2" := "OP10_384A1~Output_4_word_2";
   #IAI_Axis[X_Axis]."Output 4 word_1" := "OP10_384A1~Output_4_word_7";
   #IAI_Axis[X_Axis]."Output 4 word_2" := "OP10_384A1~Output_4_word_8";

   #IAI_Axis[X_Axis].Mode := "ModeDB".Gen;
   #IAI_Axis[X_Axis].Par.PositionWidth := 0.05;
   #IAI_Axis[X_Axis].Par.AccSpeed := 10;
   #IAI_Axis[X_Axis].Par.DecSpeed := 10;

   #IAI_Axis[X_Axis].Par."Limt+Pos" := 362000.0;
   #IAI_Axis[X_Axis].Par."Limt-Pos" := -30000.0;
   #IAI_Axis[X_Axis].Interfere := TRUE;
   #IAI_Axis[X_Axis].RunSetTime := T#20S;
   #IAI_Axis[X_Axis].Par.GoPosInterfere[0] := TRUE;
   #IAI_Axis[X_Axis].Par.GoPosInterfere[1] := TRUE;
   #IAI_Axis[X_Axis].Par.GoPosInterfere[2] := TRUE;
   #IAI_Axis[X_Axis].Par.GoPosInterfere[3] := TRUE;
   #IAI_Axis[X_Axis].Par.GoPosInterfere[4] := TRUE;
   #IAI_Axis[X_Axis].Par.GoPosInterfere[5] := TRUE;
   #IAI_Axis[X_Axis].AutoPointStart := "IAI_A2".In.iAutoStart;

   "IAI_A2".Auto.Pos[1].Pos:=#IAI_Axis[X_Axis].Par.TargetPosition[1] := "Parameter".AxisRun.Axis[6].Pos1.Position;
   "IAI_A2".Auto.Pos[1].Vel := #IAI_Axis[X_Axis].Par.TargetSpeed[1] := "Parameter".AxisRun.Axis[6].Pos1.Speed;

   "IAI_A2".Auto.Pos[2].Pos:=#IAI_Axis[X_Axis].Par.TargetPosition[2] := "Parameter".AxisRun.Axis[6].Pos2.Position;
   "IAI_A2".Auto.Pos[2].Vel :=#IAI_Axis[X_Axis].Par.TargetSpeed[2] := "Parameter".AxisRun.Axis[6].Pos2.Speed;

   "IAI_A2".Auto.Pos[3].Pos:=#IAI_Axis[X_Axis].Par.TargetPosition[3] := "Parameter".AxisRun.Axis[6].Pos3.Position;
   "IAI_A2".Auto.Pos[3].Vel :=#IAI_Axis[X_Axis].Par.TargetSpeed[3] := "Parameter".AxisRun.Axis[6].Pos3.Speed;

   "IAI_A2".Auto.Pos[4].Pos:=#IAI_Axis[X_Axis].Par.TargetPosition[4] := "Parameter".AxisRun.Axis[6].Pos4.Position;
   "IAI_A2".Auto.Pos[4].Vel :=#IAI_Axis[X_Axis].Par.TargetSpeed[4] := "Parameter".AxisRun.Axis[6].Pos4.Speed;

   "IAI_A2".Auto.Pos[5].Pos:=#IAI_Axis[X_Axis].Par.TargetPosition[5] := "Parameter".AxisRun.Axis[6].Pos5.Position;
   "IAI_A2".Auto.Pos[5].Vel :=#IAI_Axis[X_Axis].Par.TargetSpeed[5] := "Parameter".AxisRun.Axis[6].Pos5.Speed;

   "IAI_A2".Auto.Pos[6].Pos := #IAI_Axis[X_Axis].Par.TargetPosition[6] := "Parameter".AxisRun.Axis[6].Pos6.Position;
   "IAI_A2".Auto.Pos[6].Vel := #IAI_Axis[X_Axis].Par.TargetSpeed[6] := "Parameter".AxisRun.Axis[6].Pos6.Speed;

   "IAI_A2".Auto.Pos[7].Pos := #IAI_Axis[X_Axis].Par.TargetPosition[7] := "Parameter".AxisRun.Axis[6].Pos7.Position;
   "IAI_A2".Auto.Pos[7].Vel := #IAI_Axis[X_Axis].Par.TargetSpeed[7] := "Parameter".AxisRun.Axis[6].Pos7.Speed;

   "IAI_A2".Auto.Pos[8].Pos := #IAI_Axis[X_Axis].Par.TargetPosition[8] := "Parameter".AxisRun.Axis[6].Pos8.Position;
   "IAI_A2".Auto.Pos[8].Vel := #IAI_Axis[X_Axis].Par.TargetSpeed[8] := "Parameter".AxisRun.Axis[6].Pos8.Speed;

   "IAI_A2".Auto.Pos[9].Pos := #IAI_Axis[X_Axis].Par.TargetPosition[9] := "Parameter".AxisRun.Axis[6].Pos9.Position;
   "IAI_A2".Auto.Pos[9].Vel := #IAI_Axis[X_Axis].Par.TargetSpeed[9] := "Parameter".AxisRun.Axis[6].Pos9.Speed;

   "IAI_A2".Auto.Pos[10].Pos := #IAI_Axis[X_Axis].Par.TargetPosition[10] := "Parameter".AxisRun.Axis[6].Pos10.Position;
   "IAI_A2".Auto.Pos[10].Vel := #IAI_Axis[X_Axis].Par.TargetSpeed[10] := "Parameter".AxisRun.Axis[6].Pos10.Speed;

   ///Y轴
   #IAI_Axis[Y_axis]();

   #IAI_Axis[Y_axis].Axis_ID := 3;
   #IAI_Axis[Y_axis]."Input 4 word_Man1" := "OP10_384A1~Input_4_word_7";
   #IAI_Axis[Y_axis]."Input 4 word_Man2" := "OP10_384A1~Input_4_word_8";
   #IAI_Axis[Y_axis]."Input 4 word_1" := "OP10_384A1~Input_4_word_1";
   #IAI_Axis[Y_axis]."Input 4 word_2" := "OP10_384A1~Input_4_word_2";
   #IAI_Axis[Y_axis]."Output 4 word_Man1" := "OP10_384A1~Output_4_word_1";
   #IAI_Axis[Y_axis]."Output 4 word_Man2" := "OP10_384A1~Output_4_word_2";
   #IAI_Axis[Y_axis]."Output 4 word_1" := "OP10_384A1~Output_4_word_3";
   #IAI_Axis[Y_axis]."Output 4 word_2" := "OP10_384A1~Output_4_word_4";

   #IAI_Axis[Y_axis].Mode := "ModeDB".Gen;
   #IAI_Axis[Y_axis].Par.PositionWidth := 0.05;
   #IAI_Axis[Y_axis].Par.AccSpeed := 10;
   #IAI_Axis[Y_axis].Par.DecSpeed := 10;

   #IAI_Axis[Y_axis].Par."Limt+Pos" := 362000.0;
   #IAI_Axis[Y_axis].Par."Limt-Pos" := -30000.0;
   #IAI_Axis[Y_axis].Interfere := TRUE;
   #IAI_Axis[Y_axis].RunSetTime := T#20S;
   #IAI_Axis[Y_axis].Par.GoPosInterfere[0] := TRUE;
   #IAI_Axis[Y_axis].Par.GoPosInterfere[1] := TRUE;
   #IAI_Axis[Y_axis].Par.GoPosInterfere[2] := TRUE;
   #IAI_Axis[Y_axis].Par.GoPosInterfere[3] := TRUE;
   #IAI_Axis[Y_axis].Par.GoPosInterfere[4] := TRUE;
   #IAI_Axis[Y_axis].Par.GoPosInterfere[5] := TRUE;
   #IAI_Axis[Y_axis].AutoPointStart := "IAI_A3".In.iAutoStart;

   "IAI_A3".Auto.Pos[1].Pos:=#IAI_Axis[Y_axis].Par.TargetPosition[1] := "Parameter".AxisRun.Axis[7].Pos1.Position;
   "IAI_A3".Auto.Pos[1].Vel :=#IAI_Axis[Y_axis].Par.TargetSpeed[1] := "Parameter".AxisRun.Axis[7].Pos1.Speed;

   "IAI_A3".Auto.Pos[2].Pos:=#IAI_Axis[Y_axis].Par.TargetPosition[2] := "Parameter".AxisRun.Axis[7].Pos2.Position;
   "IAI_A3".Auto.Pos[2].Vel :=#IAI_Axis[Y_axis].Par.TargetSpeed[2] := "Parameter".AxisRun.Axis[7].Pos2.Speed;

   "IAI_A3".Auto.Pos[3].Pos:=#IAI_Axis[Y_axis].Par.TargetPosition[3] := "Parameter".AxisRun.Axis[7].Pos3.Position;
   "IAI_A3".Auto.Pos[3].Vel :=#IAI_Axis[Y_axis].Par.TargetSpeed[3] := "Parameter".AxisRun.Axis[7].Pos3.Speed;

   "IAI_A3".Auto.Pos[4].Pos:=#IAI_Axis[Y_axis].Par.TargetPosition[4] := "Parameter".AxisRun.Axis[7].Pos4.Position;
   "IAI_A3".Auto.Pos[4].Vel :=#IAI_Axis[Y_axis].Par.TargetSpeed[4] := "Parameter".AxisRun.Axis[7].Pos4.Speed;

   "IAI_A3".Auto.Pos[5].Pos:=#IAI_Axis[Y_axis].Par.TargetPosition[5] := "Parameter".AxisRun.Axis[7].Pos5.Position;
   "IAI_A3".Auto.Pos[5].Vel :=#IAI_Axis[Y_axis].Par.TargetSpeed[5] := "Parameter".AxisRun.Axis[7].Pos5.Speed;

   "IAI_A3".Auto.Pos[6].Pos := #IAI_Axis[Y_axis].Par.TargetPosition[6] := "Parameter".AxisRun.Axis[7].Pos6.Position;
   "IAI_A3".Auto.Pos[6].Vel := #IAI_Axis[Y_axis].Par.TargetSpeed[6] := "Parameter".AxisRun.Axis[7].Pos6.Speed;

   "IAI_A3".Auto.Pos[7].Pos := #IAI_Axis[Y_axis].Par.TargetPosition[7] := "Parameter".AxisRun.Axis[7].Pos7.Position;
   "IAI_A3".Auto.Pos[7].Vel := #IAI_Axis[Y_axis].Par.TargetSpeed[7] := "Parameter".AxisRun.Axis[7].Pos7.Speed;

   "IAI_A3".Auto.Pos[8].Pos := #IAI_Axis[Y_axis].Par.TargetPosition[8] := "Parameter".AxisRun.Axis[7].Pos8.Position;
   "IAI_A3".Auto.Pos[8].Vel := #IAI_Axis[Y_axis].Par.TargetSpeed[8] := "Parameter".AxisRun.Axis[7].Pos8.Speed;

   "IAI_A3".Auto.Pos[9].Pos := #IAI_Axis[Y_axis].Par.TargetPosition[9] := "Parameter".AxisRun.Axis[7].Pos9.Position;
   "IAI_A3".Auto.Pos[9].Vel := #IAI_Axis[Y_axis].Par.TargetSpeed[9] := "Parameter".AxisRun.Axis[7].Pos9.Speed;

   "IAI_A3".Auto.Pos[10].Pos := #IAI_Axis[Y_axis].Par.TargetPosition[10] := "Parameter".AxisRun.Axis[7].Pos10.Position;
   "IAI_A3".Auto.Pos[10].Vel := #IAI_Axis[Y_axis].Par.TargetSpeed[10] := "Parameter".AxisRun.Axis[7].Pos10.Speed;

   /////////////////HNI_DATA_PUT&GET////////
   IF "ModeDB".Gen.Out.Manual AND NOT "DB_PARAMETERS_TEACH".HMI_PAGE_CONTROL.TEACH_MODE_ACTIVE THEN
       #IAI_Axis["HMISystemDB".HMI_Axis.INPUT.Axis_ID].Par.Speed := "HMISystemDB".HMI_Axis.INPUT.Speed;
       #IAI_Axis["HMISystemDB".HMI_Axis.INPUT.Axis_ID].Par.SimplyTrigger := "HMISystemDB".HMI_Axis.INPUT.SimplyTrigger;
       #IAI_Axis["HMISystemDB".HMI_Axis.INPUT.Axis_ID].Par.SimplyTriggerPos := "HMISystemDB".HMI_Axis.INPUT.SimplyPos;
       #IAI_Axis["HMISystemDB".HMI_Axis.INPUT.Axis_ID].Par.ListTrigger := "HMISystemDB".HMI_Axis.INPUT.ListTrigger;
       #IAI_Axis["HMISystemDB".HMI_Axis.INPUT.Axis_ID].Par.ListPosID := "HMISystemDB".HMI_Axis.INPUT.ListPosID;
       #IAI_Axis["HMISystemDB".HMI_Axis.INPUT.Axis_ID].Enable := "HMISystemDB".HMI_Axis.INPUT.Enable;
       #IAI_Axis["HMISystemDB".HMI_Axis.INPUT.Axis_ID]."Jog+" := "HMISystemDB".HMI_Axis.INPUT."Jog+";
       #IAI_Axis["HMISystemDB".HMI_Axis.INPUT.Axis_ID]."Jog-" := "HMISystemDB".HMI_Axis.INPUT."Jog-";
       #IAI_Axis["HMISystemDB".HMI_Axis.INPUT.Axis_ID].Homing := "HMISystemDB".HMI_Axis.INPUT.Homing;
       #IAI_Axis["HMISystemDB".HMI_Axis.INPUT.Axis_ID].Stop := "HMISystemDB".HMI_Axis.INPUT.Stop;

     ELSIF "ModeDB".Gen.Out.Manual AND  "DB_PARAMETERS_TEACH".HMI_PAGE_CONTROL.TEACH_MODE_ACTIVE THEN

       #IAI_Axis[Z_Axis].Par.Speed := "DB_PARAMETERS_TEACH".HMI_PAGE_CONTROL.Speeds.Glue_IAI.Z;
       #IAI_Axis[Y_axis].Par.Speed := "DB_PARAMETERS_TEACH".HMI_PAGE_CONTROL.Speeds.Glue_IAI.Y;
       #IAI_Axis[X_Axis].Par.Speed := "DB_PARAMETERS_TEACH".HMI_PAGE_CONTROL.Speeds.Glue_IAI.X;


       #IAI_Axis[Z_Axis].Par.SimplyTriggerPos := "DB_PARAMETERS_TEACH".HMI_PAGE_CONTROL.Go_to_pos.Glue_IAI.Z;
       #IAI_Axis[Y_axis].Par.SimplyTriggerPos := "DB_PARAMETERS_TEACH".HMI_PAGE_CONTROL.Go_to_pos.Glue_IAI.Y;
       #IAI_Axis[X_Axis].Par.SimplyTriggerPos := "DB_PARAMETERS_TEACH".HMI_PAGE_CONTROL.Go_to_pos.Glue_IAI.X;

       #IAI_Axis[Z_Axis].Par.SimplyTrigger := "DB_PARAMETERS_TEACH".HMI_PAGE_CONTROL.Go_to_pos_TRIGGER.Glue_IAI.Z;
       #IAI_Axis[Y_axis].Par.SimplyTrigger :="DB_PARAMETERS_TEACH".HMI_PAGE_CONTROL.Go_to_pos_TRIGGER.Glue_IAI.Y ;
       #IAI_Axis[X_Axis].Par.SimplyTrigger := "DB_PARAMETERS_TEACH".HMI_PAGE_CONTROL.Go_to_pos_TRIGGER.Glue_IAI.X;


     END_IF;


   "HMISystemDB".HMI_Axis.OUTPUT.MAX_Axis := 3;
   "HMISystemDB".HMI_Axis.OUTPUT.Ready := #IAI_Axis["HMISystemDB".HMI_Axis.INPUT.Axis_ID].Ready;
   "HMISystemDB".HMI_Axis.OUTPUT.Alarm := #IAI_Axis["HMISystemDB".HMI_Axis.INPUT.Axis_ID].Error OR #IAI_Axis["HMISystemDB".HMI_Axis.INPUT.Axis_ID].OverTime;
   "HMISystemDB".HMI_Axis.OUTPUT.Warming := #IAI_Axis["HMISystemDB".HMI_Axis.INPUT.Axis_ID].Warn;
   "HMISystemDB".HMI_Axis.OUTPUT.RunEnd := #IAI_Axis["HMISystemDB".HMI_Axis.INPUT.Axis_ID].RunEnd;
   "HMISystemDB".HMI_Axis.OUTPUT.Interference := #IAI_Axis["HMISystemDB".HMI_Axis.INPUT.Axis_ID].InterfereEnable;
   "HMISystemDB".HMI_Axis.OUTPUT."Reference Point" := #IAI_Axis["HMISystemDB".HMI_Axis.INPUT.Axis_ID].Homed;
   "HMISystemDB".HMI_Axis.OUTPUT.CurrentPosition := #IAI_Axis["HMISystemDB".HMI_Axis.INPUT.Axis_ID].CurrentPosition;
   "HMISystemDB".HMI_Axis.OUTPUT.CurrentSpeed := #IAI_Axis["HMISystemDB".HMI_Axis.INPUT.Axis_ID].CurrentSpeed;
   "HMISystemDB".HMI_Axis.OUTPUT.Enable := #IAI_Axis["HMISystemDB".HMI_Axis.INPUT.Axis_ID].Enabled;
   "HMISystemDB".HMI_Axis.OUTPUT.TargetPosition := #IAI_Axis["HMISystemDB".HMI_Axis.INPUT.Axis_ID].Par.TargetPosition["HMISystemDB".HMI_Axis.INPUT.ListPosID];


   IF "ModeDB".Gen.Out.Change THEN
     #IAI_Axis[Z_Axis].Par.SimplyTriggerPos := 0.0;
     #IAI_Axis[X_Axis].Par.SimplyTriggerPos := 0.0;
     #IAI_Axis[Y_axis].Par.SimplyTriggerPos := 0.0;
       "HMISystemDB".HMI_Axis.INPUT.SimplyPos := 0.0;
   END_IF;
END_FUNCTION_BLOCK

FUNCTION_BLOCK "IAI_BASE_FB"   // FB2201, SCL
{ S7_Optimized_Access := 'FALSE' }
// stored: AutoNumber false, SetENOAutomatically false
   VAR_INPUT
      Mode : "ModeGenStruct";
      "Input 4 word_Man1" : HW_IO;
      "Input 4 word_Man2" : HW_IO;
      "Input 4 word_1" : HW_IO;
      "Input 4 word_2" : HW_IO;
      "Output 4 word_Man1" : HW_IO;
      "Output 4 word_Man2" : HW_IO;
      "Output 4 word_1" : HW_IO;
      "Output 4 word_2" : HW_IO;
      Interfere : Bool;   // 干涉条件
      Axis_ID { ExternalAccessible := 'False'; ExternalVisible := 'False'; ExternalWritable := 'False'} : Int;   // 轴编号
      AutoPointStart : Bool;
   END_VAR
   VAR_IN_OUT
      Homing : Bool;   // 回原位
      AbsPos : Bool;   // 绝对位移
      RelaPos : Bool;   // 相对位移
      Enable : Bool;   // 使能
      Stop : Bool;   // 电机停止
      "Jog+" : Bool;   // 电缸JOG+
      "Jog-" : Bool;   // 电缸JOG-
      PosCode : Int;   // 反馈位置代码
      RunEnd : Bool;   // 运行结束
      Adjist : Bool;   // 屏蔽干涉
   END_VAR
   VAR
      Par { ExternalAccessible := 'False'; ExternalVisible := 'False'; ExternalWritable := 'False'} : Struct
         "Limit+" : Bool;   // 输入的正极限
         "Limit-" : Bool;   // 输入的负极限
         PositionWidth : Real;   // 位置误差范围
         PosCode : Int;   // 位置编号
         Speed : Int;   // 速度
         "Limt+Pos" : Real;   // 软极限位置+
         "Limt-Pos" : Real;   // 软极限位置-
         AccSpeed : Int;   // 加速度
         DecSpeed : Int;   // 减速度
         LuV : Int;   // 速度倍率
         SimplyTrigger : Bool;   // 直接启动
         SimplyTriggerPos : Real;   // 直接启动位置
         ListTrigger : Bool;   // 位置列表启动
         ListPosID : Int;   // 位置列表位置ID
         TargetPosition : Array[0..30] of Real;   // 位置编号
         TargetSpeed : Array[0..30] of Int;   // 速度编号
         GoPosInterfere : Array[0..30] of Bool;   // 位置编号使能
         OverTime : Time;   // 运行时间
      END_STRUCT;
      RecvData { S7_SetPoint := 'True'} : "IAI Input Struct";
      SendData { S7_SetPoint := 'True'} : "IAI Output Struct";
      CurrentPosition : Real;   // 当前位置
      CurrentSpeed : Int;   // 当前速度
      TargetPosition : Real;   // 伺服的目标位置
      Ready : Bool;   // 私服准备好
      Enabled : Bool;   // 使能OK
      Homed : Bool;   // 相对式在原位信号
      Error : Bool;   // 电机报错
      Warn : Bool;   // 驱动器报警
      HRunning : Bool;   // 回原点运行信号
      PRunning : Bool;   // 走目标位置运行中信号
      Running : Bool;   // 运行中信号
      TemWritePos : Bool;
      TemGoPos : Bool;
      TemStart : Bool;
      RInterfere : Bool;
      PosInterfere : Bool;
      InterfereEnable : Bool;   // 干涉条件使能
      LimtStop : Bool;
      HomeJogTime { S7_SetPoint := 'True'} : TON_TIME;
      TemHomingok { S7_SetPoint := 'True'} : TON_TIME;
      TemPosOk { S7_SetPoint := 'True'} : TON_TIME;
      RunTime { S7_SetPoint := 'True'} : TON_TIME;
      RunSetTime : Time;
      OverTime : Bool;   // 运行超时报警
      Cmd : Struct
         Homing : Bool;
         PosRun : Bool;
         Jog : Bool;
      END_STRUCT;
      Hstep : Int;   // 回原点步骤
      "Step" : Int;   // 定位控制运行步骤
      PosTime { S7_SetPoint := 'True'} : TON_TIME;
      StopCmd : Bool;
      StopTime { S7_SetPoint := 'True'} : TON_TIME;
      Pos_ID : Int := 1;
      SetPosCode { S7_SetPoint := 'True'} : Int;
      AutoStart : Bool;
      TemPage { ExternalVisible := 'False'} : Int;
      TemGroup { ExternalVisible := 'False'} : Int;
      FOR_ID : Int;
      TemHMIClick : Bool;
      aRetvalRead { ExternalAccessible := 'False'; ExternalVisible := 'False'; ExternalWritable := 'False'} : Array[1..5] of Int;   // 通讯读指令的返回值
      aRetvalWrite { ExternalAccessible := 'False'; ExternalVisible := 'False'; ExternalWritable := 'False'} : Array[1..5] of Int;   // 通讯写指令的返回值
      PRunninDelay : TON_TIME;
   END_VAR
BEGIN
   //=========================================================
   //========================输入映射=========================

   REGION 伺服赋值
       // 获取网关状态
       #aRetvalRead[1] := DPRD_DAT(LADDR := #"Input 4 word_Man1", RECORD => #RecvData."Input 4 word_Man1");
       #aRetvalRead[2] := DPRD_DAT(LADDR := #"Input 4 word_Man2", RECORD => #RecvData."Input 4 word_Man2");

       // 获取轴状态
       #aRetvalRead[3] := DPRD_DAT(LADDR := #"Input 4 word_1", RECORD => #RecvData."Input 4 word_1");
       #aRetvalRead[4] := DPRD_DAT(LADDR := #"Input 4 word_2", RECORD => #RecvData."Input 4 word_2");

       #SendData."Output 4 word_2"."Accelerated Speed" := #Par.AccSpeed;  // 加速度    
   END_REGION
   REGION 电机功能检测及设定    
       ////////////网关打开/////////////
       #SendData."Output 4 word_Man1".Mon := TRUE;
       //////////////伺服报警////////////////
       IF #RecvData."Input 4 word_2".ALM OR #OverTime THEN
           #Error := true;
       END_IF;
       //////////////软极限位检测停止/////////////
       IF (#TargetPosition < #Par."Limt-Pos") OR (#TargetPosition > #Par."Limt+Pos") THEN
           #LimtStop := true;
       ELSE
           #LimtStop := false;
       END_IF;
       ///////////触碰极限位置停止伺服运行///////
       IF #LimtStop OR #Par."Limit+" OR #Par."Limit-" THEN
           #Step := 0;
           #Hstep := 0;
           #AbsPos := false;
           #RelaPos := false;
       END_IF;
       //////////////伺服报错终止运行///////////////
       IF NOT #Mode.Out.Estop OR #RecvData."Input 4 word_2".ALM = TRUE THEN
           #Hstep := 0;
           #Step := 0;
           #SendData."Output 4 word_2".STP := TRUE;
           #Homing := false;
           #TemStart := false;
       END_IF;
       ///////////////模式变化///////////////////
       IF #Mode.Out.Change THEN
           #SetPosCode := #Par.PosCode;
           #Par.PosCode := #PosCode;
           #"Jog-" := false;
           #"Jog+" := false;
           #Homing := false;
           #AbsPos := false;
           #RelaPos := false;
           #Step := 0;
           #Hstep := 0;
       END_IF;
       /////////位置代码干涉条件判断//////////////
       IF #Par.ListTrigger OR #TemGoPos THEN

           IF #Par.GoPosInterfere[#Par.PosCode] THEN
               #PosInterfere := true;
           ELSE
               #PosInterfere := false;
           END_IF;
       ELSE
           #PosInterfere := true;
       END_IF;
       #RInterfere := #PosInterfere AND #Interfere;
       ////////////干涉条件判断/////////////////////
       IF #RInterfere OR #Adjist THEN
           #InterfereEnable := true;
       ELSE
           #InterfereEnable := false;
       END_IF;
       //////////////轴使能//////////   
       IF #Mode.Out.Estop AND #RecvData."Input 4 word_2".ALM = FALSE AND #Enable THEN //((#Mode.Out.Manual AND #Enable) OR #Mode.Out.Auto)
           #SendData."Output 4 word_2".SON := TRUE;
       ELSE
           #SendData."Output 4 word_2".SON := FALSE;
       END_IF;
       ////////////使能反馈/////////////
       IF #SendData."Output 4 word_2".SON AND #Mode.Out.Estop THEN
           #Enabled := true;
       ELSE
           #Enabled := false;
       END_IF;
       ///////////轴报错初始化步骤/////////////
       IF #Error THEN
           #Step := 0;
           #"Jog-" := false;
           #"Jog+" := false;
           #Hstep := 0;
           #Homing := false;
           #TemStart := false;
       END_IF;
       ////////////复位轴报警/////////

       IF #Mode.Out.Reset THEN
           #Error := false;
           #OverTime := FALSE;
           #SendData."Output 4 word_2".RES := true;
           #SendData."Output 4 word_2".Home := FALSE;
           #Hstep := 0;
           #SendData."Output 4 word_2".STP := FALSE;
           //#SetPosCode := #Par.PosCode;
       ELSE
           #SendData."Output 4 word_2".RES := false;
       END_IF;
       //////////////Reday/////////////
       IF #Enabled AND NOT #PRunning AND #Homed AND #InterfereEnable THEN
           #Ready := true;
       ELSE
           #Ready := false;
       END_IF;
       /////////////////获取电机参数//////////////////////////
       #"CurrentPosition" := DINT_TO_REAL(IN := #RecvData."Input 4 word_1"."Current Position") / 100;
       #"CurrentSpeed" := #RecvData."Input 4 word_2"."Current Speed";
       /////////////////电机速率设置/////////////
       #SendData."Output 4 word_2".JVEL := TRUE;
       #SendData."Output 4 word_1"."Location Width" := REAL_TO_DINT(IN := (#Par.PositionWidth * 100)); //宽度。
   END_REGION
   REGION 位置判断
       IF #Mode.Out.Manual THEN
           #FOR_ID := 0;
       ELSE
           #FOR_ID := 1;
       END_IF;

       FOR #Pos_ID := #FOR_ID TO 29 DO
           IF #CurrentPosition >= #Par.TargetPosition[#Pos_ID] - #Par.PositionWidth AND
               #CurrentPosition <= #Par.TargetPosition[#Pos_ID] + #Par.PositionWidth AND #Homed THEN
               #PosCode := #Pos_ID;
               #SetPosCode := #Pos_ID;
               EXIT;
           ELSE
               #PosCode := -9;
           END_IF;
       END_FOR;

   END_REGION
   REGION 回原位
       #TemHomingok(IN := #RecvData."Input 4 word_2".Hend AND #HRunning,    //原位ok时间
                    PT := t#2s);
       //////////////////执行程序////////////    
       CASE #Hstep OF
           0:
               #HRunning := false;
               IF #Homing AND #Enabled AND #InterfereEnable THEN
                   #SendData."Output 4 word_2".Home := TRUE;
                   #Step := 0;
                   #Homed := false;
                   #Hstep := 1;
               END_IF;
           1:  // Start Homing
               IF (#RecvData."Input 4 word_2".Move = TRUE)
               THEN
                   #HRunning := true;
                   #Hstep := 2;
               END_IF;

           2:  // Home End
               IF (#RecvData."Input 4 word_2".Hend = TRUE AND #TemHomingok.Q)
               THEN
                   #SendData."Output 4 word_2".Home := FALSE;
                   #Hstep := 3;
               END_IF;

           3:  // End of Chain
               IF #SendData."Output 4 word_2".Home = FALSE THEN
                   #Homing := FALSE;
                   #Homed := TRUE;
                   #HRunning := FALSE;
                   #Hstep := 0;
               END_IF;

       END_CASE;
   END_REGION
   REGION 定位控制 
       /////////自动模式切换位置编号自动触发电机运行//////////  
       //IF #Par.PosCode <> #SetPosCode THEN
           IF (#Mode.Out.Auto OR #Mode.Out.Home) AND  #AutoPointStart THEN
               #AutoStart := TRUE;
           ELSE
               #AutoStart := false;
           END_IF;
       //END_IF;

       IF #Mode.Out.Manual AND #Par.SimplyTrigger THEN
           #Par.PosCode := 0;
           #SetPosCode := #Par.PosCode;
       ELSIF #Mode.Out.Manual AND #Par.ListTrigger THEN
           #TargetPosition := #Par.TargetPosition[#Par.ListPosID];
           #Par.PosCode := #Par.ListPosID;
           #SetPosCode := #Par.PosCode;
       END_IF;

       #Par.TargetPosition[0] := #Par.SimplyTriggerPos;
       #Par.TargetSpeed[0] := #Par.Speed;

       IF #Mode.Out.Auto THEN
           #TargetPosition := #Par.TargetPosition[#Par.PosCode];
           #SendData."Output 4 word_1"."Target position" := REAL_TO_DINT(IN := (#TargetPosition * 100));//写入目标位置
           #SendData."Output 4 word_2".Speed :=#Par.TargetSpeed[#Par.PosCode]; // 速度 
       END_IF;
       IF #Mode.Out.Manual THEN

           #SendData."Output 4 word_1"."Target position" := REAL_TO_DINT(IN := (#TargetPosition * 100));//写入目标位置
           #SendData."Output 4 word_2".Speed := #Par.Speed;//#Par.TargetSpeed[#Par.ListPosID]; // 速度 
       END_IF;
   (*    IF #Mode.Out.Manual AND #Par.PosCode = 0 THEN
           #SendData."Output 4 word_2".Speed := #Par.TargetSpeed[0]; // 速度
       ELSE
           #SendData."Output 4 word_2".Speed := #Par.TargetSpeed[#Pos_ID]; // 速度 
       END_IF; *)
       //////////////////////触发启动/////////////
       IF ((#Mode.Out.Manual AND (#Par.SimplyTrigger OR #Par.ListTrigger) AND #InterfereEnable AND #Par.Speed > 1.0))   // AND  #Par.PosCode = 0
           OR ((#Mode.Out.Auto OR #Mode.Out.Home) AND #AutoStart AND #Mode.Out.Running AND #InterfereEnable AND #Par.Speed > 1.0) THEN
           #TemStart := TRUE;
       END_IF;

       CASE #Step OF
           0:///////////////准备/////////////////// 
               #PRunning := false;
               #TemWritePos := false;
               IF #TemStart AND #Ready AND #InterfereEnable THEN
                   #SendData."Output 4 word_2".STP := FALSE;
                   #RunEnd := false;
                   #"Jog-" := false;
                   #"Jog+" := false;
                   #Step := 1;
               END_IF;
           1://////////////目标位置//////////////////   
               #PRunning := true;
               IF #TemStart THEN       //定位位置
                   #TargetPosition := #Par.TargetPosition[#Par.PosCode];
               END_IF;
               IF #TargetPosition = #Par.TargetPosition[#Par.PosCode] THEN
                   #SendData."Output 4 word_1"."Target position" := REAL_TO_DINT(IN := (#TargetPosition * 100));//写入目标位置
                   #SendData."Output 4 word_2".Speed := #Par.TargetSpeed[#Par.PosCode]; // 速度 
                   IF #TargetPosition = #CurrentPosition THEN
                       #PosCode := #Par.PosCode;
                       #PRunning := FALSE;
                       #TemStart := false;
                       #RunEnd := TRUE;
                       #SetPosCode := #Par.PosCode;
                       IF #SetPosCode = #Par.PosCode THEN
                           #Step := 0;
                       END_IF;
                   ELSE
                       #Step := 2;
                   END_IF;
               END_IF;

           2: ///////////////启动///////////////////
               #SendData."Output 4 word_1"."Target position" := REAL_TO_DINT(IN := (#TargetPosition * 100));//写入目标位置
               #SendData."Output 4 word_2".Speed := #Par.TargetSpeed[#Par.PosCode]; // 速度 
               IF #RecvData."Input 4 word_2".Pend AND "ClockMemory0.5s" AND #InterfereEnable THEN
                   #SendData."Output 4 word_2".CSTR := TRUE;
               ELSE
                   #SendData."Output 4 word_2".CSTR := FALSE;
               END_IF;
               IF #RecvData."Input 4 word_2".Pend = FALSE AND #RecvData."Input 4 word_2".Move THEN //OR #TemPosOk.Q
                   #Step := 3;
               END_IF;

           3: ///////////////////中间停止//////////////////
               IF #Stop OR #InterfereEnable = FALSE THEN
                   #StopCmd := true;
                   #SendData."Output 4 word_2".STP := TRUE;
               ELSE
                   #StopCmd := false;
                   #SendData."Output 4 word_2".STP := FALSE;
               END_IF;
               ////////////运行完成////////////////
               IF #RecvData."Input 4 word_2".Pend THEN
                   #SendData."Output 4 word_2".CSTR := FALSE;
                   #Step := 4;
               END_IF;
           4: //////位置比较////////////
               IF #Mode.Out.Manual THEN

                   IF "IAI_DeviceCtl".IAIServo[#Axis_ID].Point[#Par.ListPosID].Achieve THEN
                       #SetPosCode := #Par.PosCode;
                       IF #SetPosCode = #Par.PosCode THEN
                           ;
                           #Step := 5;
                       END_IF;
                   END_IF;
                   IF #RecvData."Input 4 word_1"."Current Position" = REAL_TO_DINT(IN := (#Par.SimplyTriggerPos * 100)) THEN
                       #Step := 5;
                   END_IF;
               END_IF;
               IF #Mode.Out.Auto THEN
                   IF "IAI_DeviceCtl".IAIServo[#Axis_ID].Point[#Par.PosCode].Achieve THEN
                       #SetPosCode := #Par.PosCode;
                       IF #SetPosCode = #Par.PosCode THEN
                           ;
                           #Step := 5;
                       END_IF;
                   END_IF;
               END_IF;
           5:
               #SendData."Output 4 word_2".CSTR := FALSE;
               #AutoStart := FALSE;
               IF #SendData."Output 4 word_2".CSTR = FALSE AND #AutoStart = FALSE THEN
                   #RunEnd := true;
                   #PRunning := false;
                   #TemStart := FALSE;
                   #Step := 0;
               END_IF;

       END_CASE;
   END_REGION
   ///////////////////////////运行时间///////////////////////
   #Running := #HRunning OR #PRunning;
   #RunTime(IN := #Running,
            PT := #RunSetTime);
   IF #RunTime.Q THEN
       #OverTime := TRUE;
   END_IF;
   ///////////////////JOG//////////////////
   REGION 点动控制
       IF #Mode.Out.Manual AND #Step = 0 THEN
           ;

           // #SendData.JISL := #"Jog+" OR #"Jog-";
           /////////////////jog+////////////////
           #SendData."Output 4 word_2"."JOG+" := #"Jog+" AND NOT #Par."Limit+" AND (#CurrentPosition < #Par."Limt+Pos");
           /////////////////jog-///////////////
           #SendData."Output 4 word_2"."JOG-" := #"Jog-" AND NOT #Par."Limit-" AND (#CurrentPosition > #Par."Limt-Pos");
       END_IF;
   END_REGION

   //==========================================================
   //=========================输出映射=========================
   //==========================================================

   //网关控制
   #aRetvalWrite[1] := DPWR_DAT(LADDR := #"Output 4 word_Man1", RECORD := #SendData."Output 4 word_Man1");
   #aRetvalWrite[2] := DPWR_DAT(LADDR := #"Output 4 word_Man2", RECORD := #SendData."Output 4 word_Man2");

   //轴控制
   #aRetvalWrite[3] := DPWR_DAT(LADDR := #"Output 4 word_1", RECORD := #SendData."Output 4 word_1");
   #aRetvalWrite[4] := DPWR_DAT(LADDR := #"Output 4 word_2", RECORD := #SendData."Output 4 word_2");
END_FUNCTION_BLOCK

FUNCTION "KistlerPresser_Main" : Void   // FC2300, LAD
{ S7_Optimized_Access := 'TRUE' }
// stored: AutoNumber false, SetENOAutomatically false
   VAR_TEMP
      tRel : DInt;
   END_VAR
   VAR_TEMP   // added for the SCL form of the ladder/FBD networks
      _w1 : Bool;
   END_VAR
BEGIN

REGION Network 1: OP10_372A1 Kistler Press
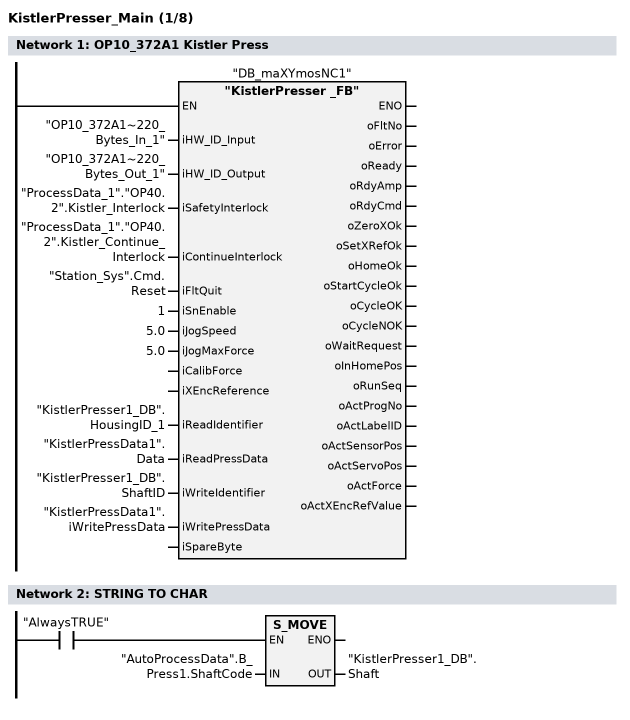
   RUNG wire#powerrail
      "DB_maXYmosNC1"(iHW_ID_Input := "OP10_372A1~220_Bytes_In_1", iHW_ID_Output := "OP10_372A1~220_Bytes_Out_1", iSafetyInterlock := "ProcessData_1"."OP40.2".Kistler_Interlock, iContinueInterlock := "ProcessData_1"."OP40.2".Kistler_Continue_Interlock, iFltQuit := "Station_Sys".Cmd.Reset, iSnEnable := 1, iJogSpeed := 5.0, iJogMaxForce := 5.0, iCalibForce :=, iXEncReference :=, iReadIdentifier := "KistlerPresser1_DB".HousingID_1, iReadPressData := "KistlerPressData1".Data, iWriteIdentifier := "KistlerPresser1_DB".ShaftID, iWritePressData := "KistlerPressData1".iWritePressData, iSpareByte :=, oFltNo =>, oError =>, oReady =>, oRdyAmp =>, oRdyCmd =>, oZeroXOk =>, oSetXRefOk =>, oHomeOk =>, oStartCycleOk =>, oCycleOK =>, oCycleNOK =>, oWaitRequest =>, oInHomePos =>, oRunSeq =>, oActProgNo =>, oActLabelID =>, oActSensorPos =>, oActServoPos =>, oActForce =>, oActXEncRefValue =>)
   END_RUNG
   // the same network as SCL:
   "DB_maXYmosNC1"(iHW_ID_Input := "OP10_372A1~220_Bytes_In_1",   // "KistlerPresser _FB"
                   iHW_ID_Output := "OP10_372A1~220_Bytes_Out_1",
                   iSafetyInterlock := "ProcessData_1"."OP40.2".Kistler_Interlock,
                   iContinueInterlock := "ProcessData_1"."OP40.2".Kistler_Continue_Interlock,
                   iFltQuit := "Station_Sys".Cmd.Reset,
                   iSnEnable := 1,
                   iJogSpeed := 5.0,
                   iJogMaxForce := 5.0,
                   iReadIdentifier := "KistlerPresser1_DB".HousingID_1,
                   iReadPressData := "KistlerPressData1".Data,
                   iWriteIdentifier := "KistlerPresser1_DB".ShaftID,
                   iWritePressData := "KistlerPressData1".iWritePressData);
END_REGION

REGION Network 2: STRING TO CHAR
   RUNG wire#powerrail
      Contact( "AlwaysTRUE" )
      S_Move(in := "AutoProcessData".B_Press1.ShaftCode, out => "KistlerPresser1_DB".Shaft)
   END_RUNG
   // the same network as SCL:
   IF "AlwaysTRUE" THEN "KistlerPresser1_DB".Shaft := "AutoProcessData".B_Press1.ShaftCode; END_IF;
END_REGION

REGION Network 3 (SCL): STRING TO CHAR
   Strg_TO_Chars(Strg:="KistlerPresser1_DB".Shaft,
                 pChars:=0,
                 Cnt=>#tRel,
                 Chars:="KistlerPresser1_DB".ShaftID);
END_REGION

REGION Network 4: OP10_372A1 Kistler Press_Safety_Interlock
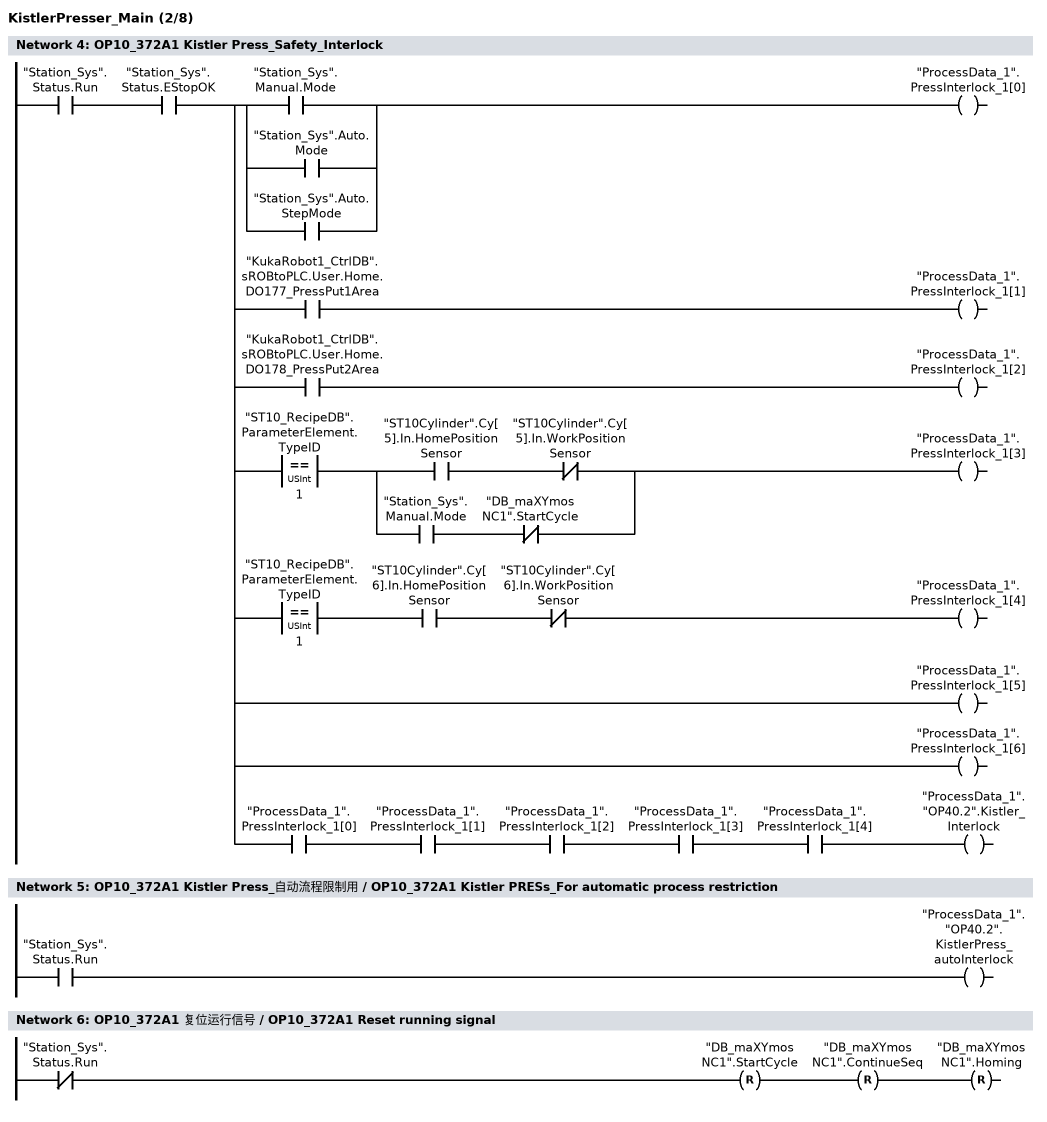
   RUNG wire#powerrail
      Contact( "Station_Sys".Status.Run )
      Contact( "Station_Sys".Status.EStopOK )
      wire#w1
      Contact( "Station_Sys".Manual.Mode )
      wire#w2
      Coil( "ProcessData_1".PressInterlock_1[0] )
   END_RUNG
   RUNG wire#w1
      Contact( "Station_Sys".Auto.Mode )
   END_RUNG wire#w2
   RUNG wire#w1
      Contact( "Station_Sys".Auto.StepMode )
   END_RUNG wire#w2
   RUNG wire#w1
      Contact( "KukaRobot1_CtrlDB".sROBtoPLC.User.Home.DO177_PressPut1Area )
      Coil( "ProcessData_1".PressInterlock_1[1] )
   END_RUNG
   RUNG wire#w1
      Contact( "KukaRobot1_CtrlDB".sROBtoPLC.User.Home.DO178_PressPut2Area )
      Coil( "ProcessData_1".PressInterlock_1[2] )
   END_RUNG
   RUNG wire#w1
      { S7_Templates := "SrcType := USInt" } EQ_Contact(in1 := "ST10_RecipeDB".ParameterElement.TypeID, in2 := 1)
      wire#w3
      Contact( "ST10Cylinder".Cy[5].In.HomePositionSensor )
      I_Contact( "ST10Cylinder".Cy[5].In.WorkPositionSensor )
      wire#w4
      Coil( "ProcessData_1".PressInterlock_1[3] )
   END_RUNG
   RUNG wire#w3
      Contact( "Station_Sys".Manual.Mode )
      I_Contact( "DB_maXYmosNC1".StartCycle )
   END_RUNG wire#w4
   RUNG wire#w1
      { S7_Templates := "SrcType := USInt" } EQ_Contact(in1 := "ST10_RecipeDB".ParameterElement.TypeID, in2 := 1)
      Contact( "ST10Cylinder".Cy[6].In.HomePositionSensor )
      I_Contact( "ST10Cylinder".Cy[6].In.WorkPositionSensor )
      Coil( "ProcessData_1".PressInterlock_1[4] )
   END_RUNG
   RUNG wire#w1
      Coil( "ProcessData_1".PressInterlock_1[5] )
   END_RUNG
   RUNG wire#w1
      Coil( "ProcessData_1".PressInterlock_1[6] )
   END_RUNG
   RUNG wire#w1
      Contact( "ProcessData_1".PressInterlock_1[0] )
      Contact( "ProcessData_1".PressInterlock_1[1] )
      Contact( "ProcessData_1".PressInterlock_1[2] )
      Contact( "ProcessData_1".PressInterlock_1[3] )
      Contact( "ProcessData_1".PressInterlock_1[4] )
      Coil( "ProcessData_1"."OP40.2".Kistler_Interlock )
   END_RUNG
   // the same network as SCL:
   #_w1 := "Station_Sys".Status.Run AND "Station_Sys".Status.EStopOK;
   "ProcessData_1".PressInterlock_1[0] := #_w1 AND ("Station_Sys".Manual.Mode OR "Station_Sys".Auto.Mode OR "Station_Sys".Auto.StepMode);
   "ProcessData_1".PressInterlock_1[1] := #_w1 AND "KukaRobot1_CtrlDB".sROBtoPLC.User.Home.DO177_PressPut1Area;
   "ProcessData_1".PressInterlock_1[2] := #_w1 AND "KukaRobot1_CtrlDB".sROBtoPLC.User.Home.DO178_PressPut2Area;
   "ProcessData_1".PressInterlock_1[3] := #_w1 AND ("ST10_RecipeDB".ParameterElement.TypeID = 1) AND (("ST10Cylinder".Cy[5].In.HomePositionSensor AND NOT "ST10Cylinder".Cy[5].In.WorkPositionSensor) OR ("Station_Sys".Manual.Mode AND NOT "DB_maXYmosNC1".StartCycle));
   "ProcessData_1".PressInterlock_1[4] := #_w1 AND ("ST10_RecipeDB".ParameterElement.TypeID = 1) AND "ST10Cylinder".Cy[6].In.HomePositionSensor AND NOT "ST10Cylinder".Cy[6].In.WorkPositionSensor;
   "ProcessData_1".PressInterlock_1[5] := #_w1;
   "ProcessData_1".PressInterlock_1[6] := #_w1;
   "ProcessData_1"."OP40.2".Kistler_Interlock := #_w1 AND "ProcessData_1".PressInterlock_1[0] AND "ProcessData_1".PressInterlock_1[1] AND "ProcessData_1".PressInterlock_1[2] AND "ProcessData_1".PressInterlock_1[3] AND "ProcessData_1".PressInterlock_1[4];
END_REGION

REGION Network 5: OP10_372A1 Kistler Press_自动流程限制用 / OP10_372A1 Kistler PRESs_For automatic process restriction
   RUNG wire#powerrail
      Contact( "Station_Sys".Status.Run )
      Coil( "ProcessData_1"."OP40.2".KistlerPress_autoInterlock )
   END_RUNG
   // the same network as SCL:
   "ProcessData_1"."OP40.2".KistlerPress_autoInterlock := "Station_Sys".Status.Run;
END_REGION

REGION Network 6: OP10_372A1 复位运行信号 / OP10_372A1 Reset running signal
   RUNG wire#powerrail
      I_Contact( "Station_Sys".Status.Run )
      R_Coil( "DB_maXYmosNC1".StartCycle )
      R_Coil( "DB_maXYmosNC1".ContinueSeq )
      R_Coil( "DB_maXYmosNC1".Homing )
   END_RUNG
   // the same network as SCL:
   IF NOT "Station_Sys".Status.Run THEN
       "DB_maXYmosNC1".StartCycle := FALSE;
       "DB_maXYmosNC1".ContinueSeq := FALSE;
       "DB_maXYmosNC1".Homing := FALSE;
   END_IF;
END_REGION

REGION Network 7: 手动模式程序号赋值 / Manual mode program number assignment
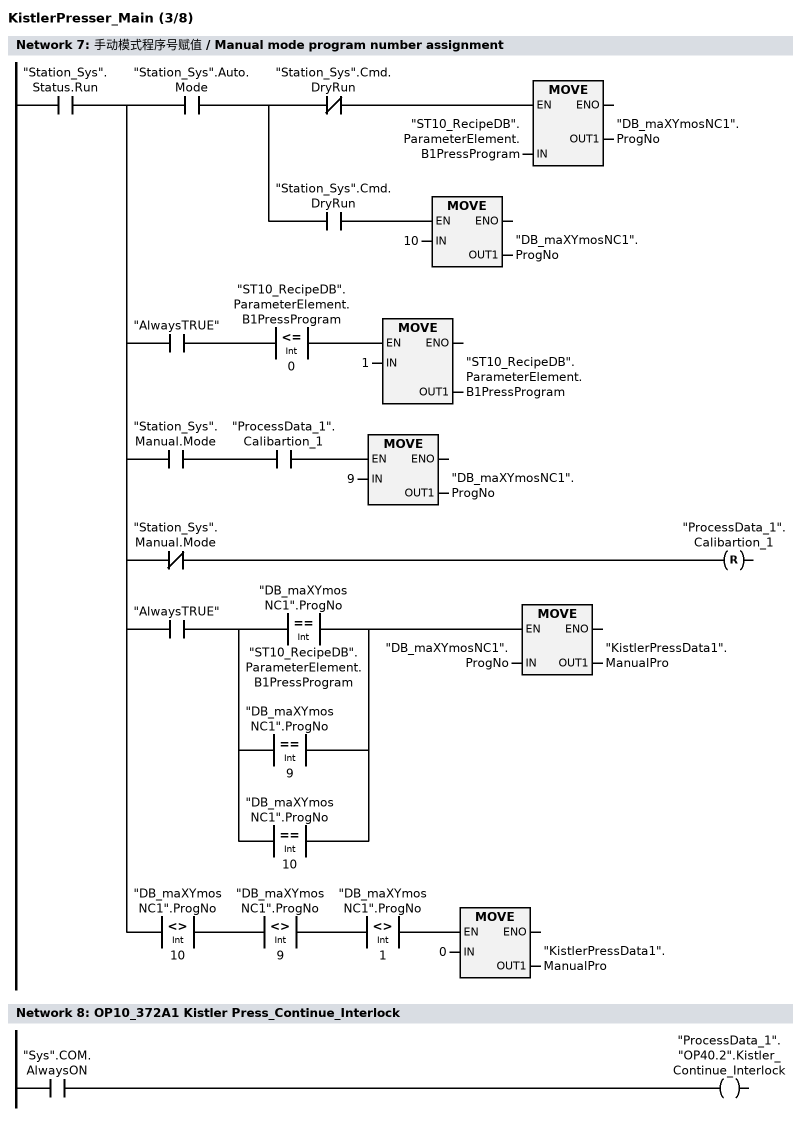
   RUNG wire#powerrail
      Contact( "Station_Sys".Status.Run )
      wire#w1
      Contact( "Station_Sys".Auto.Mode )
      wire#w2
      I_Contact( "Station_Sys".Cmd.DryRun )
      Move(in := "ST10_RecipeDB".ParameterElement.B1PressProgram, out1 => "DB_maXYmosNC1".ProgNo)
   END_RUNG
   RUNG wire#w2
      Contact( "Station_Sys".Cmd.DryRun )
      Move(in := 10, out1 => "DB_maXYmosNC1".ProgNo)
   END_RUNG
   RUNG wire#w1
      Contact( "AlwaysTRUE" )
      { S7_Templates := "SrcType := Int" } LE_Contact(in1 := "ST10_RecipeDB".ParameterElement.B1PressProgram, in2 := 0)
      Move(in := 1, out1 => "ST10_RecipeDB".ParameterElement.B1PressProgram)
   END_RUNG
   RUNG wire#w1
      Contact( "Station_Sys".Manual.Mode )
      Contact( "ProcessData_1".Calibartion_1 )
      Move(in := 9, out1 => "DB_maXYmosNC1".ProgNo)
   END_RUNG
   RUNG wire#w1
      I_Contact( "Station_Sys".Manual.Mode )
      R_Coil( "ProcessData_1".Calibartion_1 )
   END_RUNG
   RUNG wire#w1
      Contact( "AlwaysTRUE" )
      wire#w3
      { S7_Templates := "SrcType := Int" } EQ_Contact(in1 := "DB_maXYmosNC1".ProgNo, in2 := "ST10_RecipeDB".ParameterElement.B1PressProgram)
      wire#w4
      Move(in := "DB_maXYmosNC1".ProgNo, out1 => "KistlerPressData1".ManualPro)
   END_RUNG
   RUNG wire#w3
      { S7_Templates := "SrcType := Int" } EQ_Contact(in1 := "DB_maXYmosNC1".ProgNo, in2 := 9)
   END_RUNG wire#w4
   RUNG wire#w3
      { S7_Templates := "SrcType := Int" } EQ_Contact(in1 := "DB_maXYmosNC1".ProgNo, in2 := 10)
   END_RUNG wire#w4
   RUNG wire#w1
      { S7_Templates := "SrcType := Int" } NE_Contact(in1 := "DB_maXYmosNC1".ProgNo, in2 := 10)
      { S7_Templates := "SrcType := Int" } NE_Contact(in1 := "DB_maXYmosNC1".ProgNo, in2 := 9)
      { S7_Templates := "SrcType := Int" } NE_Contact(in1 := "DB_maXYmosNC1".ProgNo, in2 := 1)
      Move(in := 0, out1 => "KistlerPressData1".ManualPro)
   END_RUNG
   // the same network as SCL:
   #_w1 := "Station_Sys".Status.Run AND "Station_Sys".Auto.Mode;
   IF #_w1 AND NOT "Station_Sys".Cmd.DryRun THEN
       "DB_maXYmosNC1".ProgNo := "ST10_RecipeDB".ParameterElement.B1PressProgram;
   END_IF;
   IF #_w1 AND "Station_Sys".Cmd.DryRun THEN "DB_maXYmosNC1".ProgNo := 10; END_IF;
   IF "Station_Sys".Status.Run AND "AlwaysTRUE" AND ("ST10_RecipeDB".ParameterElement.B1PressProgram <= 0) THEN
       "ST10_RecipeDB".ParameterElement.B1PressProgram := 1;
   END_IF;
   IF "Station_Sys".Status.Run AND "Station_Sys".Manual.Mode AND "ProcessData_1".Calibartion_1 THEN
       "DB_maXYmosNC1".ProgNo := 9;
   END_IF;
   IF "Station_Sys".Status.Run AND NOT "Station_Sys".Manual.Mode THEN
       "ProcessData_1".Calibartion_1 := FALSE;
   END_IF;
   IF "Station_Sys".Status.Run AND "AlwaysTRUE" AND (("DB_maXYmosNC1".ProgNo = "ST10_RecipeDB".ParameterElement.B1PressProgram) OR ("DB_maXYmosNC1".ProgNo = 9) OR ("DB_maXYmosNC1".ProgNo = 10)) THEN
       "KistlerPressData1".ManualPro := "DB_maXYmosNC1".ProgNo;
   END_IF;
   IF "Station_Sys".Status.Run AND ("DB_maXYmosNC1".ProgNo <> 10) AND ("DB_maXYmosNC1".ProgNo <> 9) AND ("DB_maXYmosNC1".ProgNo <> 1) THEN
       "KistlerPressData1".ManualPro := 0;
   END_IF;
END_REGION

REGION Network 8: OP10_372A1 Kistler Press_Continue_Interlock
   RUNG wire#powerrail
      Contact( "Sys".COM.AlwaysON )
      Coil( "ProcessData_1"."OP40.2".Kistler_Continue_Interlock )
   END_RUNG
   // the same network as SCL:
   "ProcessData_1"."OP40.2".Kistler_Continue_Interlock := "Sys".COM.AlwaysON;
END_REGION

REGION Network 9: OP10_372A1 KistlerPressData 奇石乐第1次压装数据 / OP10_372A1 KistlerPressData The first KistlerPressdata
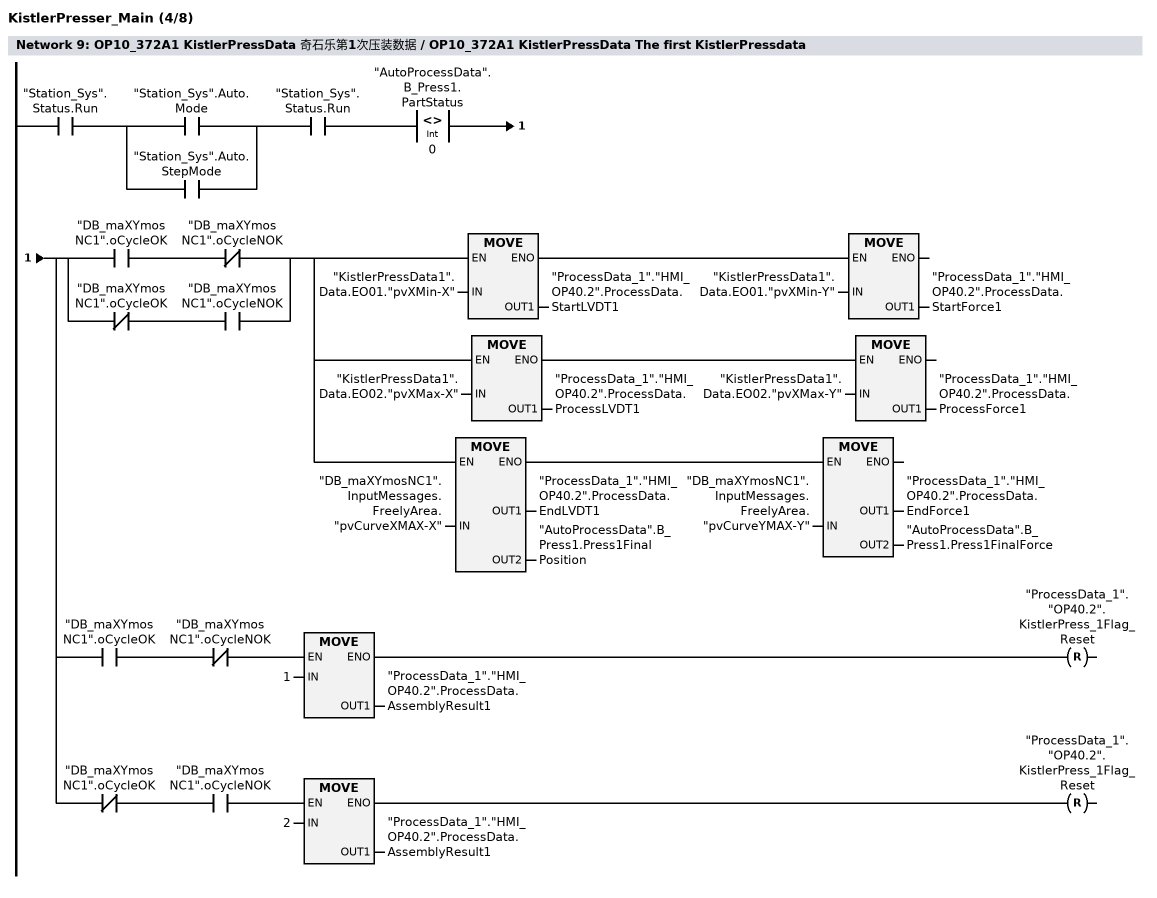
   RUNG wire#powerrail
      Contact( "Station_Sys".Status.Run )
      wire#w1
      Contact( "Station_Sys".Auto.Mode )
      wire#w2
      Contact( "Station_Sys".Status.Run )
      { S7_Templates := "SrcType := Int" } NE_Contact(in1 := "AutoProcessData".B_Press1.PartStatus, in2 := 0)
      wire#w3
      Contact( "DB_maXYmosNC1".oCycleOK )
      I_Contact( "DB_maXYmosNC1".oCycleNOK )
      wire#w4
      Move(in := "KistlerPressData1".Data.EO01."pvXMin-X", out1 => "ProcessData_1"."HMI_OP40.2".ProcessData.StartLVDT1)
      Move(in := "KistlerPressData1".Data.EO01."pvXMin-Y", out1 => "ProcessData_1"."HMI_OP40.2".ProcessData.StartForce1)
   END_RUNG
   RUNG wire#w1
      Contact( "Station_Sys".Auto.StepMode )
   END_RUNG wire#w2
   RUNG wire#w3
      I_Contact( "DB_maXYmosNC1".oCycleOK )
      Contact( "DB_maXYmosNC1".oCycleNOK )
   END_RUNG wire#w4
   RUNG wire#w4
      Move(in := "KistlerPressData1".Data.EO02."pvXMax-X", out1 => "ProcessData_1"."HMI_OP40.2".ProcessData.ProcessLVDT1)
      Move(in := "KistlerPressData1".Data.EO02."pvXMax-Y", out1 => "ProcessData_1"."HMI_OP40.2".ProcessData.ProcessForce1)
   END_RUNG
   RUNG wire#w4
      Move(in := "DB_maXYmosNC1".InputMessages.FreelyArea."pvCurveXMAX-X", out1 => "ProcessData_1"."HMI_OP40.2".ProcessData.EndLVDT1, out2 => "AutoProcessData".B_Press1.Press1FinalPosition)
      Move(in := "DB_maXYmosNC1".InputMessages.FreelyArea."pvCurveYMAX-Y", out1 => "ProcessData_1"."HMI_OP40.2".ProcessData.EndForce1, out2 => "AutoProcessData".B_Press1.Press1FinalForce)
   END_RUNG
   RUNG wire#w3
      Contact( "DB_maXYmosNC1".oCycleOK )
      I_Contact( "DB_maXYmosNC1".oCycleNOK )
      Move(in := 1, out1 => "ProcessData_1"."HMI_OP40.2".ProcessData.AssemblyResult1)
      R_Coil( "ProcessData_1"."OP40.2".KistlerPress_1Flag_Reset )
   END_RUNG
   RUNG wire#w3
      I_Contact( "DB_maXYmosNC1".oCycleOK )
      Contact( "DB_maXYmosNC1".oCycleNOK )
      Move(in := 2, out1 => "ProcessData_1"."HMI_OP40.2".ProcessData.AssemblyResult1)
      R_Coil( "ProcessData_1"."OP40.2".KistlerPress_1Flag_Reset )
   END_RUNG
   // the same network as SCL:
   #_w1 := "Station_Sys".Status.Run AND ("Station_Sys".Auto.Mode OR "Station_Sys".Auto.StepMode) AND "Station_Sys".Status.Run AND ("AutoProcessData".B_Press1.PartStatus <> 0);
   IF #_w1 AND (("DB_maXYmosNC1".oCycleOK AND NOT "DB_maXYmosNC1".oCycleNOK) OR (NOT "DB_maXYmosNC1".oCycleOK AND "DB_maXYmosNC1".oCycleNOK)) THEN
       "ProcessData_1"."HMI_OP40.2".ProcessData.StartLVDT1 := "KistlerPressData1".Data.EO01."pvXMin-X";
       "ProcessData_1"."HMI_OP40.2".ProcessData.StartForce1 := "KistlerPressData1".Data.EO01."pvXMin-Y";
       "ProcessData_1"."HMI_OP40.2".ProcessData.ProcessLVDT1 := "KistlerPressData1".Data.EO02."pvXMax-X";
       "ProcessData_1"."HMI_OP40.2".ProcessData.ProcessForce1 := "KistlerPressData1".Data.EO02."pvXMax-Y";
       "ProcessData_1"."HMI_OP40.2".ProcessData.EndLVDT1 := "DB_maXYmosNC1".InputMessages.FreelyArea."pvCurveXMAX-X";
       "AutoProcessData".B_Press1.Press1FinalPosition := "DB_maXYmosNC1".InputMessages.FreelyArea."pvCurveXMAX-X";
       "ProcessData_1"."HMI_OP40.2".ProcessData.EndForce1 := "DB_maXYmosNC1".InputMessages.FreelyArea."pvCurveYMAX-Y";
       "AutoProcessData".B_Press1.Press1FinalForce := "DB_maXYmosNC1".InputMessages.FreelyArea."pvCurveYMAX-Y";
   END_IF;
   IF #_w1 AND "DB_maXYmosNC1".oCycleOK AND NOT "DB_maXYmosNC1".oCycleNOK THEN
       "ProcessData_1"."HMI_OP40.2".ProcessData.AssemblyResult1 := 1;
       "ProcessData_1"."OP40.2".KistlerPress_1Flag_Reset := FALSE;
   END_IF;
   IF #_w1 AND NOT "DB_maXYmosNC1".oCycleOK AND "DB_maXYmosNC1".oCycleNOK THEN
       "ProcessData_1"."HMI_OP40.2".ProcessData.AssemblyResult1 := 2;
       "ProcessData_1"."OP40.2".KistlerPress_1Flag_Reset := FALSE;
   END_IF;
END_REGION

REGION Network 11: OP10_375A1 Kistler Press
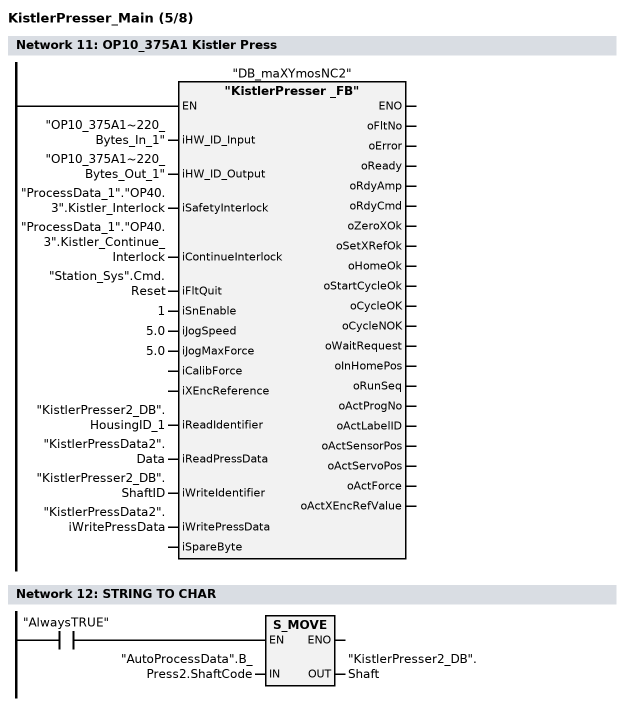
   RUNG wire#powerrail
      "DB_maXYmosNC2"(iHW_ID_Input := "OP10_375A1~220_Bytes_In_1", iHW_ID_Output := "OP10_375A1~220_Bytes_Out_1", iSafetyInterlock := "ProcessData_1"."OP40.3".Kistler_Interlock, iContinueInterlock := "ProcessData_1"."OP40.3".Kistler_Continue_Interlock, iFltQuit := "Station_Sys".Cmd.Reset, iSnEnable := 1, iJogSpeed := 5.0, iJogMaxForce := 5.0, iCalibForce :=, iXEncReference :=, iReadIdentifier := "KistlerPresser2_DB".HousingID_1, iReadPressData := "KistlerPressData2".Data, iWriteIdentifier := "KistlerPresser2_DB".ShaftID, iWritePressData := "KistlerPressData2".iWritePressData, iSpareByte :=, oFltNo =>, oError =>, oReady =>, oRdyAmp =>, oRdyCmd =>, oZeroXOk =>, oSetXRefOk =>, oHomeOk =>, oStartCycleOk =>, oCycleOK =>, oCycleNOK =>, oWaitRequest =>, oInHomePos =>, oRunSeq =>, oActProgNo =>, oActLabelID =>, oActSensorPos =>, oActServoPos =>, oActForce =>, oActXEncRefValue =>)
   END_RUNG
   // the same network as SCL:
   "DB_maXYmosNC2"(iHW_ID_Input := "OP10_375A1~220_Bytes_In_1",   // "KistlerPresser _FB"
                   iHW_ID_Output := "OP10_375A1~220_Bytes_Out_1",
                   iSafetyInterlock := "ProcessData_1"."OP40.3".Kistler_Interlock,
                   iContinueInterlock := "ProcessData_1"."OP40.3".Kistler_Continue_Interlock,
                   iFltQuit := "Station_Sys".Cmd.Reset,
                   iSnEnable := 1,
                   iJogSpeed := 5.0,
                   iJogMaxForce := 5.0,
                   iReadIdentifier := "KistlerPresser2_DB".HousingID_1,
                   iReadPressData := "KistlerPressData2".Data,
                   iWriteIdentifier := "KistlerPresser2_DB".ShaftID,
                   iWritePressData := "KistlerPressData2".iWritePressData);
END_REGION

REGION Network 12: STRING TO CHAR
   RUNG wire#powerrail
      Contact( "AlwaysTRUE" )
      S_Move(in := "AutoProcessData".B_Press2.ShaftCode, out => "KistlerPresser2_DB".Shaft)
   END_RUNG
   // the same network as SCL:
   IF "AlwaysTRUE" THEN "KistlerPresser2_DB".Shaft := "AutoProcessData".B_Press2.ShaftCode; END_IF;
END_REGION

REGION Network 13 (SCL): STRING TO CHAR
   Strg_TO_Chars(Strg:="KistlerPresser2_DB".Shaft,
                 pChars:=0,
                 Cnt=>#tRel,
                 Chars:="KistlerPresser2_DB".ShaftID);
END_REGION

REGION Network 14: OP10_375A1 Kistler Press_Safety_Interlock
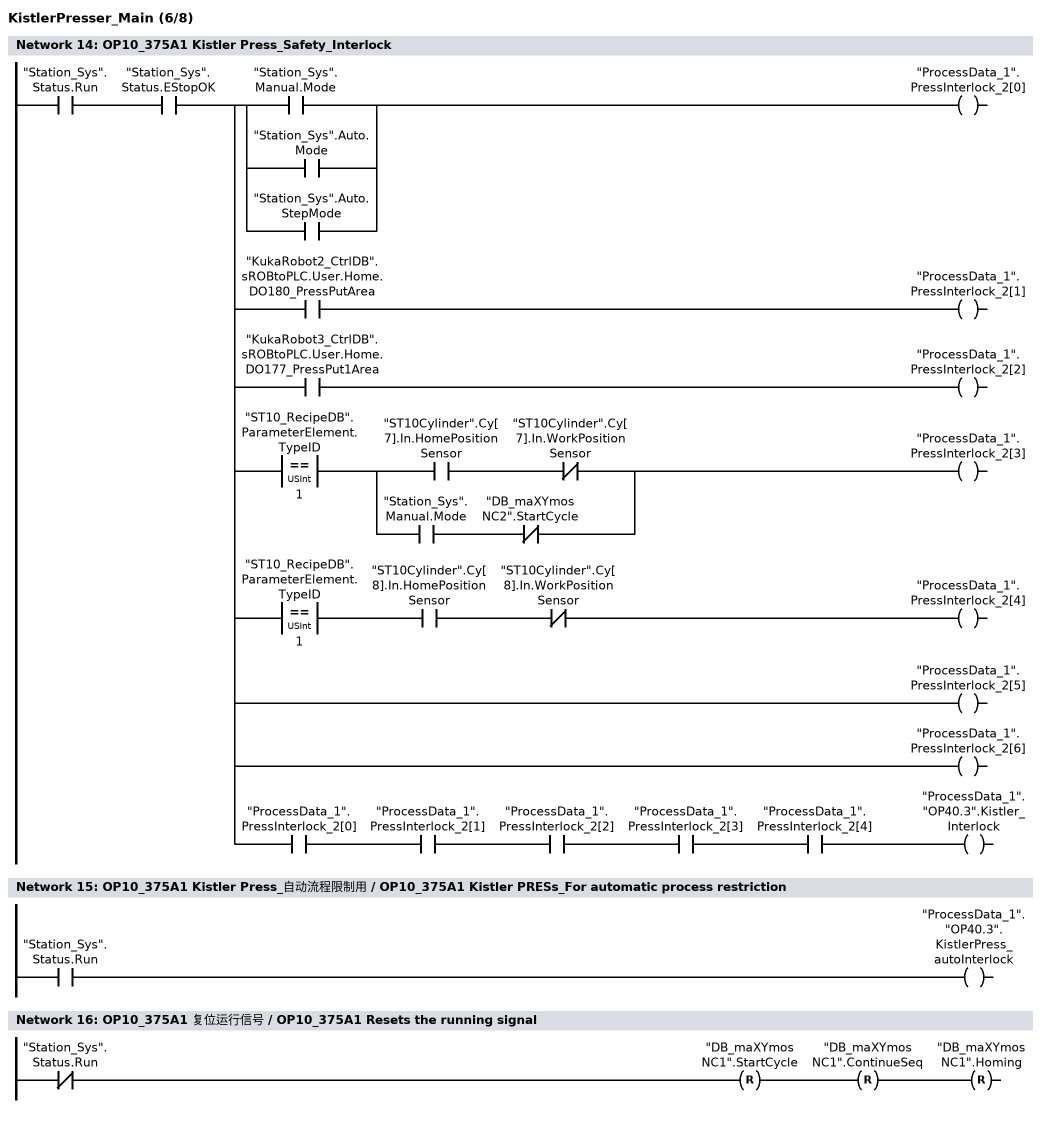
   RUNG wire#powerrail
      Contact( "Station_Sys".Status.Run )
      Contact( "Station_Sys".Status.EStopOK )
      wire#w1
      Contact( "Station_Sys".Manual.Mode )
      wire#w2
      Coil( "ProcessData_1".PressInterlock_2[0] )
   END_RUNG
   RUNG wire#w1
      Contact( "Station_Sys".Auto.Mode )
   END_RUNG wire#w2
   RUNG wire#w1
      Contact( "Station_Sys".Auto.StepMode )
   END_RUNG wire#w2
   RUNG wire#w1
      Contact( "KukaRobot2_CtrlDB".sROBtoPLC.User.Home.DO180_PressPutArea )
      Coil( "ProcessData_1".PressInterlock_2[1] )
   END_RUNG
   RUNG wire#w1
      Contact( "KukaRobot3_CtrlDB".sROBtoPLC.User.Home.DO177_PressPut1Area )
      Coil( "ProcessData_1".PressInterlock_2[2] )
   END_RUNG
   RUNG wire#w1
      { S7_Templates := "SrcType := USInt" } EQ_Contact(in1 := "ST10_RecipeDB".ParameterElement.TypeID, in2 := 1)
      wire#w3
      Contact( "ST10Cylinder".Cy[7].In.HomePositionSensor )
      I_Contact( "ST10Cylinder".Cy[7].In.WorkPositionSensor )
      wire#w4
      Coil( "ProcessData_1".PressInterlock_2[3] )
   END_RUNG
   RUNG wire#w3
      Contact( "Station_Sys".Manual.Mode )
      I_Contact( "DB_maXYmosNC2".StartCycle )
   END_RUNG wire#w4
   RUNG wire#w1
      { S7_Templates := "SrcType := USInt" } EQ_Contact(in1 := "ST10_RecipeDB".ParameterElement.TypeID, in2 := 1)
      Contact( "ST10Cylinder".Cy[8].In.HomePositionSensor )
      I_Contact( "ST10Cylinder".Cy[8].In.WorkPositionSensor )
      Coil( "ProcessData_1".PressInterlock_2[4] )
   END_RUNG
   RUNG wire#w1
      Coil( "ProcessData_1".PressInterlock_2[5] )
   END_RUNG
   RUNG wire#w1
      Coil( "ProcessData_1".PressInterlock_2[6] )
   END_RUNG
   RUNG wire#w1
      Contact( "ProcessData_1".PressInterlock_2[0] )
      Contact( "ProcessData_1".PressInterlock_2[1] )
      Contact( "ProcessData_1".PressInterlock_2[2] )
      Contact( "ProcessData_1".PressInterlock_2[3] )
      Contact( "ProcessData_1".PressInterlock_2[4] )
      Coil( "ProcessData_1"."OP40.3".Kistler_Interlock )
   END_RUNG
   // the same network as SCL:
   #_w1 := "Station_Sys".Status.Run AND "Station_Sys".Status.EStopOK;
   "ProcessData_1".PressInterlock_2[0] := #_w1 AND ("Station_Sys".Manual.Mode OR "Station_Sys".Auto.Mode OR "Station_Sys".Auto.StepMode);
   "ProcessData_1".PressInterlock_2[1] := #_w1 AND "KukaRobot2_CtrlDB".sROBtoPLC.User.Home.DO180_PressPutArea;
   "ProcessData_1".PressInterlock_2[2] := #_w1 AND "KukaRobot3_CtrlDB".sROBtoPLC.User.Home.DO177_PressPut1Area;
   "ProcessData_1".PressInterlock_2[3] := #_w1 AND ("ST10_RecipeDB".ParameterElement.TypeID = 1) AND (("ST10Cylinder".Cy[7].In.HomePositionSensor AND NOT "ST10Cylinder".Cy[7].In.WorkPositionSensor) OR ("Station_Sys".Manual.Mode AND NOT "DB_maXYmosNC2".StartCycle));
   "ProcessData_1".PressInterlock_2[4] := #_w1 AND ("ST10_RecipeDB".ParameterElement.TypeID = 1) AND "ST10Cylinder".Cy[8].In.HomePositionSensor AND NOT "ST10Cylinder".Cy[8].In.WorkPositionSensor;
   "ProcessData_1".PressInterlock_2[5] := #_w1;
   "ProcessData_1".PressInterlock_2[6] := #_w1;
   "ProcessData_1"."OP40.3".Kistler_Interlock := #_w1 AND "ProcessData_1".PressInterlock_2[0] AND "ProcessData_1".PressInterlock_2[1] AND "ProcessData_1".PressInterlock_2[2] AND "ProcessData_1".PressInterlock_2[3] AND "ProcessData_1".PressInterlock_2[4];
END_REGION

REGION Network 15: OP10_375A1 Kistler Press_自动流程限制用 / OP10_375A1 Kistler PRESs_For automatic process restriction
   RUNG wire#powerrail
      Contact( "Station_Sys".Status.Run )
      Coil( "ProcessData_1"."OP40.3".KistlerPress_autoInterlock )
   END_RUNG
   // the same network as SCL:
   "ProcessData_1"."OP40.3".KistlerPress_autoInterlock := "Station_Sys".Status.Run;
END_REGION

REGION Network 16: OP10_375A1 复位运行信号 / OP10_375A1 Resets the running signal
   RUNG wire#powerrail
      I_Contact( "Station_Sys".Status.Run )
      R_Coil( "DB_maXYmosNC1".StartCycle )
      R_Coil( "DB_maXYmosNC1".ContinueSeq )
      R_Coil( "DB_maXYmosNC1".Homing )
   END_RUNG
   // the same network as SCL:
   IF NOT "Station_Sys".Status.Run THEN
       "DB_maXYmosNC1".StartCycle := FALSE;
       "DB_maXYmosNC1".ContinueSeq := FALSE;
       "DB_maXYmosNC1".Homing := FALSE;
   END_IF;
END_REGION

REGION Network 17: 手动模式程序号赋值 / Manual mode program number assignment
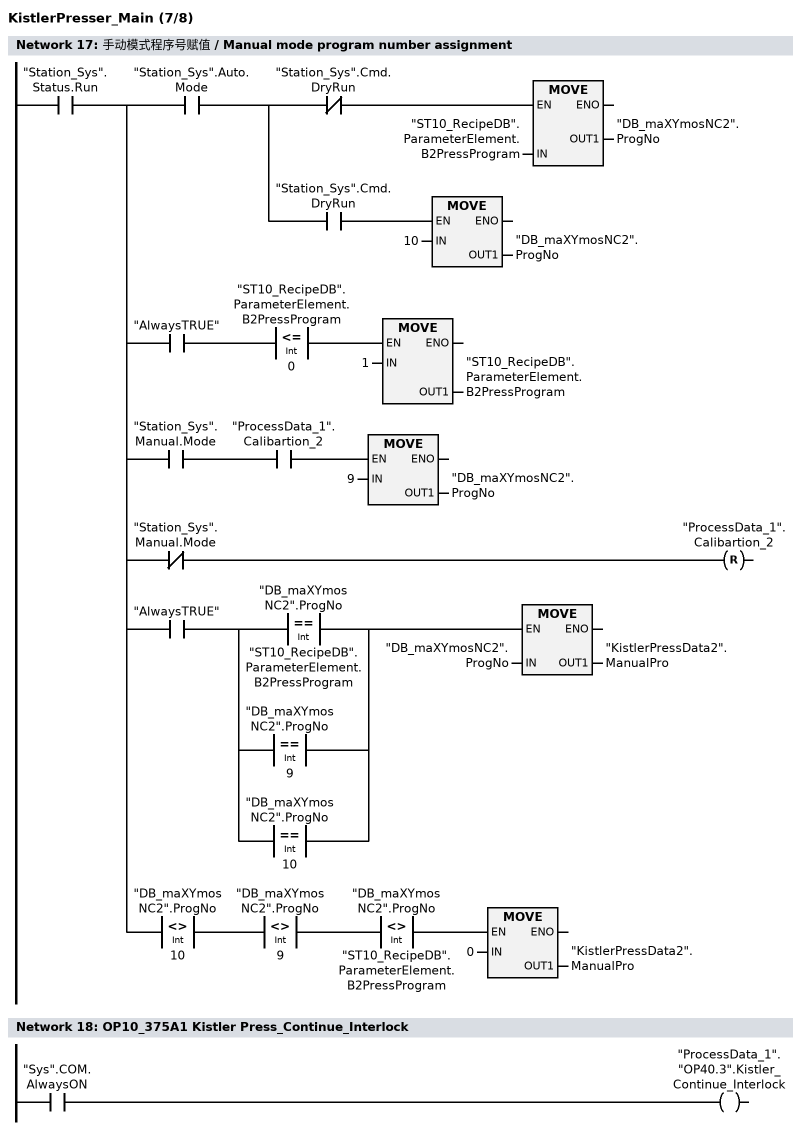
   RUNG wire#powerrail
      Contact( "Station_Sys".Status.Run )
      wire#w1
      Contact( "Station_Sys".Auto.Mode )
      wire#w2
      I_Contact( "Station_Sys".Cmd.DryRun )
      Move(in := "ST10_RecipeDB".ParameterElement.B2PressProgram, out1 => "DB_maXYmosNC2".ProgNo)
   END_RUNG
   RUNG wire#w2
      Contact( "Station_Sys".Cmd.DryRun )
      Move(in := 10, out1 => "DB_maXYmosNC2".ProgNo)
   END_RUNG
   RUNG wire#w1
      Contact( "AlwaysTRUE" )
      { S7_Templates := "SrcType := Int" } LE_Contact(in1 := "ST10_RecipeDB".ParameterElement.B2PressProgram, in2 := 0)
      Move(in := 1, out1 => "ST10_RecipeDB".ParameterElement.B2PressProgram)
   END_RUNG
   RUNG wire#w1
      Contact( "Station_Sys".Manual.Mode )
      Contact( "ProcessData_1".Calibartion_2 )
      Move(in := 9, out1 => "DB_maXYmosNC2".ProgNo)
   END_RUNG
   RUNG wire#w1
      I_Contact( "Station_Sys".Manual.Mode )
      R_Coil( "ProcessData_1".Calibartion_2 )
   END_RUNG
   RUNG wire#w1
      Contact( "AlwaysTRUE" )
      wire#w3
      { S7_Templates := "SrcType := Int" } EQ_Contact(in1 := "DB_maXYmosNC2".ProgNo, in2 := "ST10_RecipeDB".ParameterElement.B2PressProgram)
      wire#w4
      Move(in := "DB_maXYmosNC2".ProgNo, out1 => "KistlerPressData2".ManualPro)
   END_RUNG
   RUNG wire#w3
      { S7_Templates := "SrcType := Int" } EQ_Contact(in1 := "DB_maXYmosNC2".ProgNo, in2 := 9)
   END_RUNG wire#w4
   RUNG wire#w3
      { S7_Templates := "SrcType := Int" } EQ_Contact(in1 := "DB_maXYmosNC2".ProgNo, in2 := 10)
   END_RUNG wire#w4
   RUNG wire#w1
      { S7_Templates := "SrcType := Int" } NE_Contact(in1 := "DB_maXYmosNC2".ProgNo, in2 := 10)
      { S7_Templates := "SrcType := Int" } NE_Contact(in1 := "DB_maXYmosNC2".ProgNo, in2 := 9)
      { S7_Templates := "SrcType := Int" } NE_Contact(in1 := "DB_maXYmosNC2".ProgNo, in2 := "ST10_RecipeDB".ParameterElement.B2PressProgram)
      Move(in := 0, out1 => "KistlerPressData2".ManualPro)
   END_RUNG
   // the same network as SCL:
   #_w1 := "Station_Sys".Status.Run AND "Station_Sys".Auto.Mode;
   IF #_w1 AND NOT "Station_Sys".Cmd.DryRun THEN
       "DB_maXYmosNC2".ProgNo := "ST10_RecipeDB".ParameterElement.B2PressProgram;
   END_IF;
   IF #_w1 AND "Station_Sys".Cmd.DryRun THEN "DB_maXYmosNC2".ProgNo := 10; END_IF;
   IF "Station_Sys".Status.Run AND "AlwaysTRUE" AND ("ST10_RecipeDB".ParameterElement.B2PressProgram <= 0) THEN
       "ST10_RecipeDB".ParameterElement.B2PressProgram := 1;
   END_IF;
   IF "Station_Sys".Status.Run AND "Station_Sys".Manual.Mode AND "ProcessData_1".Calibartion_2 THEN
       "DB_maXYmosNC2".ProgNo := 9;
   END_IF;
   IF "Station_Sys".Status.Run AND NOT "Station_Sys".Manual.Mode THEN
       "ProcessData_1".Calibartion_2 := FALSE;
   END_IF;
   IF "Station_Sys".Status.Run AND "AlwaysTRUE" AND (("DB_maXYmosNC2".ProgNo = "ST10_RecipeDB".ParameterElement.B2PressProgram) OR ("DB_maXYmosNC2".ProgNo = 9) OR ("DB_maXYmosNC2".ProgNo = 10)) THEN
       "KistlerPressData2".ManualPro := "DB_maXYmosNC2".ProgNo;
   END_IF;
   IF "Station_Sys".Status.Run AND ("DB_maXYmosNC2".ProgNo <> 10) AND ("DB_maXYmosNC2".ProgNo <> 9) AND ("DB_maXYmosNC2".ProgNo <> "ST10_RecipeDB".ParameterElement.B2PressProgram) THEN
       "KistlerPressData2".ManualPro := 0;
   END_IF;
END_REGION

REGION Network 18: OP10_375A1 Kistler Press_Continue_Interlock
   RUNG wire#powerrail
      Contact( "Sys".COM.AlwaysON )
      Coil( "ProcessData_1"."OP40.3".Kistler_Continue_Interlock )
   END_RUNG
   // the same network as SCL:
   "ProcessData_1"."OP40.3".Kistler_Continue_Interlock := "Sys".COM.AlwaysON;
END_REGION

REGION Network 19: OP10_375A1 KistlerPressData 奇石乐第1次压装数据 / OP10_375A1 KistlerPressData The first KistlerPressdata
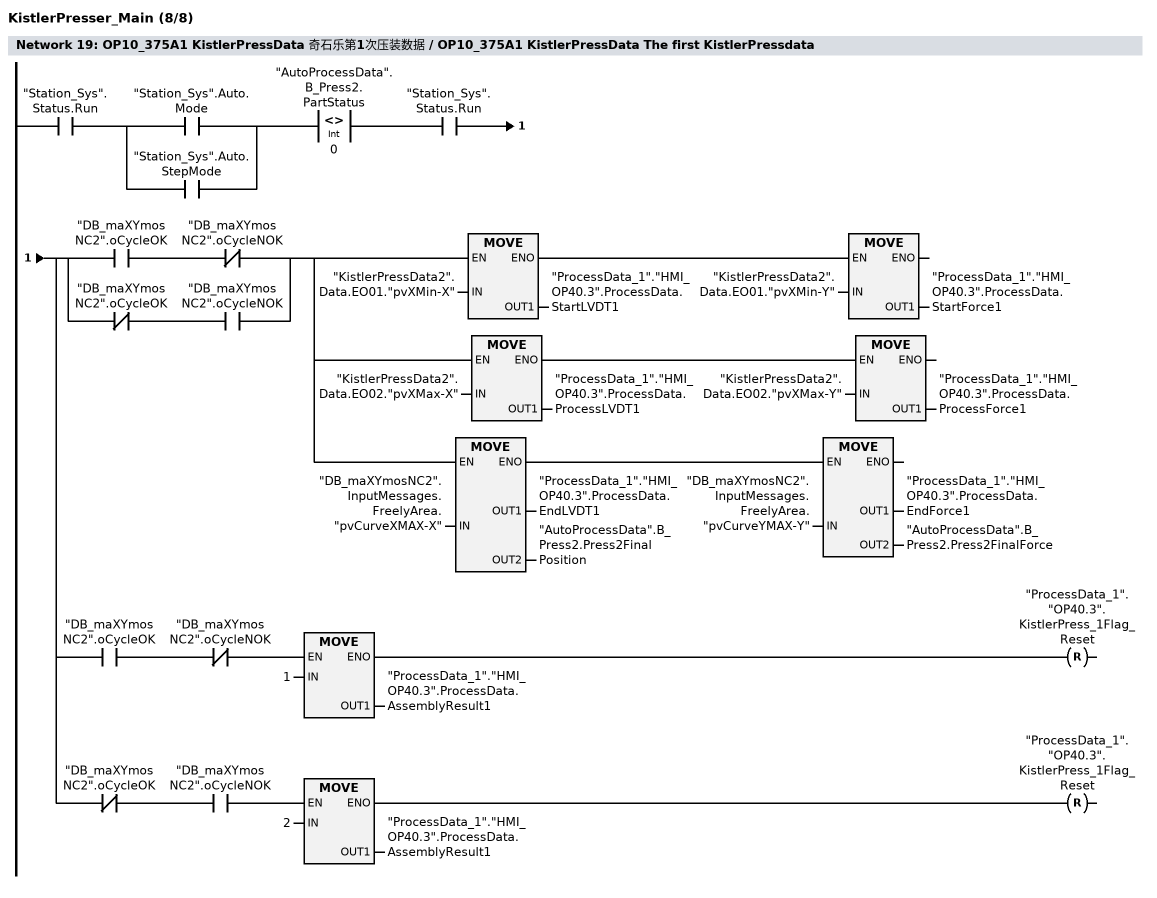
   RUNG wire#powerrail
      Contact( "Station_Sys".Status.Run )
      wire#w1
      Contact( "Station_Sys".Auto.Mode )
      wire#w2
      { S7_Templates := "SrcType := Int" } NE_Contact(in1 := "AutoProcessData".B_Press2.PartStatus, in2 := 0)
      Contact( "Station_Sys".Status.Run )
      wire#w3
      Contact( "DB_maXYmosNC2".oCycleOK )
      I_Contact( "DB_maXYmosNC2".oCycleNOK )
      wire#w4
      Move(in := "KistlerPressData2".Data.EO01."pvXMin-X", out1 => "ProcessData_1"."HMI_OP40.3".ProcessData.StartLVDT1)
      Move(in := "KistlerPressData2".Data.EO01."pvXMin-Y", out1 => "ProcessData_1"."HMI_OP40.3".ProcessData.StartForce1)
   END_RUNG
   RUNG wire#w1
      Contact( "Station_Sys".Auto.StepMode )
   END_RUNG wire#w2
   RUNG wire#w3
      I_Contact( "DB_maXYmosNC2".oCycleOK )
      Contact( "DB_maXYmosNC2".oCycleNOK )
   END_RUNG wire#w4
   RUNG wire#w4
      Move(in := "KistlerPressData2".Data.EO02."pvXMax-X", out1 => "ProcessData_1"."HMI_OP40.3".ProcessData.ProcessLVDT1)
      Move(in := "KistlerPressData2".Data.EO02."pvXMax-Y", out1 => "ProcessData_1"."HMI_OP40.3".ProcessData.ProcessForce1)
   END_RUNG
   RUNG wire#w4
      Move(in := "DB_maXYmosNC2".InputMessages.FreelyArea."pvCurveXMAX-X", out1 => "ProcessData_1"."HMI_OP40.3".ProcessData.EndLVDT1, out2 => "AutoProcessData".B_Press2.Press2FinalPosition)
      Move(in := "DB_maXYmosNC2".InputMessages.FreelyArea."pvCurveYMAX-Y", out1 => "ProcessData_1"."HMI_OP40.3".ProcessData.EndForce1, out2 => "AutoProcessData".B_Press2.Press2FinalForce)
   END_RUNG
   RUNG wire#w3
      Contact( "DB_maXYmosNC2".oCycleOK )
      I_Contact( "DB_maXYmosNC2".oCycleNOK )
      Move(in := 1, out1 => "ProcessData_1"."HMI_OP40.3".ProcessData.AssemblyResult1)
      R_Coil( "ProcessData_1"."OP40.3".KistlerPress_1Flag_Reset )
   END_RUNG
   RUNG wire#w3
      I_Contact( "DB_maXYmosNC2".oCycleOK )
      Contact( "DB_maXYmosNC2".oCycleNOK )
      Move(in := 2, out1 => "ProcessData_1"."HMI_OP40.3".ProcessData.AssemblyResult1)
      R_Coil( "ProcessData_1"."OP40.3".KistlerPress_1Flag_Reset )
   END_RUNG
   // the same network as SCL:
   #_w1 := "Station_Sys".Status.Run AND ("Station_Sys".Auto.Mode OR "Station_Sys".Auto.StepMode) AND ("AutoProcessData".B_Press2.PartStatus <> 0) AND "Station_Sys".Status.Run;
   IF #_w1 AND (("DB_maXYmosNC2".oCycleOK AND NOT "DB_maXYmosNC2".oCycleNOK) OR (NOT "DB_maXYmosNC2".oCycleOK AND "DB_maXYmosNC2".oCycleNOK)) THEN
       "ProcessData_1"."HMI_OP40.3".ProcessData.StartLVDT1 := "KistlerPressData2".Data.EO01."pvXMin-X";
       "ProcessData_1"."HMI_OP40.3".ProcessData.StartForce1 := "KistlerPressData2".Data.EO01."pvXMin-Y";
       "ProcessData_1"."HMI_OP40.3".ProcessData.ProcessLVDT1 := "KistlerPressData2".Data.EO02."pvXMax-X";
       "ProcessData_1"."HMI_OP40.3".ProcessData.ProcessForce1 := "KistlerPressData2".Data.EO02."pvXMax-Y";
       "ProcessData_1"."HMI_OP40.3".ProcessData.EndLVDT1 := "DB_maXYmosNC2".InputMessages.FreelyArea."pvCurveXMAX-X";
       "AutoProcessData".B_Press2.Press2FinalPosition := "DB_maXYmosNC2".InputMessages.FreelyArea."pvCurveXMAX-X";
       "ProcessData_1"."HMI_OP40.3".ProcessData.EndForce1 := "DB_maXYmosNC2".InputMessages.FreelyArea."pvCurveYMAX-Y";
       "AutoProcessData".B_Press2.Press2FinalForce := "DB_maXYmosNC2".InputMessages.FreelyArea."pvCurveYMAX-Y";
   END_IF;
   IF #_w1 AND "DB_maXYmosNC2".oCycleOK AND NOT "DB_maXYmosNC2".oCycleNOK THEN
       "ProcessData_1"."HMI_OP40.3".ProcessData.AssemblyResult1 := 1;
       "ProcessData_1"."OP40.3".KistlerPress_1Flag_Reset := FALSE;
   END_IF;
   IF #_w1 AND NOT "DB_maXYmosNC2".oCycleOK AND "DB_maXYmosNC2".oCycleNOK THEN
       "ProcessData_1"."HMI_OP40.3".ProcessData.AssemblyResult1 := 2;
       "ProcessData_1"."OP40.3".KistlerPress_1Flag_Reset := FALSE;
   END_IF;
END_REGION
END_FUNCTION

